  MoveL 2939 to (264.24, 330.75, -7.5) mm, rotated rx 180 ry 0 rz -180 deg; joints [-12.648, -42.636, 107.245, 166.05, 65.267, -174.067]
  MoveL 2940 to (259.09, 331.49, -7.5) mm, rotated rx 180 ry 0 rz 180 deg; joints [-12.718, -42.745, 107.572, 165.997, 65.486, -174.093]
  MoveL 2941 to (253.9, 331.91, -7.5) mm, rotated rx -180 ry 0 rz 180 deg; joints [-12.777, -42.855, 107.905, 165.957, 65.708, -174.125]
  MoveL 2942 to (248.7, 331.99, -7.5) mm, rotated rx -180 ry 0 rz -180 deg; joints [-12.824, -42.967, 108.243, 165.931, 65.932, -174.164]
  MoveL 2943 to (243.5, 331.74, -7.5) mm, rotated rx -180 ry 0 rz 180 deg; joints [-12.859, -43.079, 108.585, 165.917, 66.159, -174.21]
  MoveL 2944 to (238.33, 331.17, -7.5) mm, rotated rx -180 ry 0 rz -180 deg; joints [-12.882, -43.192, 108.929, 165.917, 66.386, -174.262]
  MoveL 2945 to (233.21, 330.26, -7.5) mm, rotated rx 180 ry 0 rz 180 deg; joints [-12.892, -43.304, 109.274, 165.931, 66.613, -174.319]
  MoveL 2946 to (228.15, 329.04, -7.5) mm, rotated rx -180 ry 0 rz 180 deg; joints [-12.89, -43.415, 109.619, 165.958, 66.839, -174.382]
  MoveL 2947 to (223.18, 327.49, -7.5) mm, rotated rx -180 ry 0 rz -180 deg; joints [-12.874, -43.525, 109.963, 165.999, 67.064, -174.45]
  MoveL 2948 to (218.32, 325.63, -7.5) mm, rotated rx 180 ry 0 rz -180 deg; joints [-12.846, -43.634, 110.303, 166.053, 67.286, -174.523]
  MoveL 2949 to (213.59, 323.47, -7.5) mm, rotated rx 180 ry 0 rz -180 deg; joints [-12.804, -43.741, 110.638, 166.121, 67.504, -174.599]
  MoveL 2950 to (209, 321.01, -7.5) mm, rotated rx 180 ry 0 rz 180 deg; joints [-12.75, -43.845, 110.968, 166.202, 67.718, -174.68]
  MoveL 2951 to (204.58, 318.27, -7.5) mm, rotated rx -180 ry 0 rz 180 deg; joints [-12.683, -43.946, 111.291, 166.296, 67.927, -174.764]
  MoveL 2952 to (200.34, 315.25, -7.5) mm, rotated rx -180 ry 0 rz -180 deg; joints [-12.603, -44.044, 111.605, 166.402, 68.13, -174.851]
  MoveL 2953 to (196.3, 311.97, -7.5) mm, rotated rx 180 ry 0 rz 180 deg; joints [-12.51, -44.138, 111.909, 166.521, 68.326, -174.941]
  MoveL 2954 to (192.48, 308.44, -7.5) mm, rotated rx -180 ry 0 rz 180 deg; joints [-12.406, -44.228, 112.202, 166.651, 68.515, -175.033]
  MoveL 2955 to (188.89, 304.68, -7.5) mm, rotated rx -180 ry 0 rz 180 deg; joints [-12.29, -44.314, 112.483, 166.793, 68.694, -175.126]
  MoveL 2956 to (185.54, 300.69, -7.5) mm, rotated rx -180 ry 0 rz -180 deg; joints [-12.162, -44.395, 112.751, 166.946, 68.865, -175.221]
  MoveL 2957 to (182.46, 296.5, -7.5) mm, rotated rx -180 ry 0 rz 180 deg; joints [-12.023, -44.472, 113.004, 167.11, 69.025, -175.317]
  MoveL 2958 to (179.65, 292.12, -7.5) mm, rotated rx 180 ry 0 rz -180 deg; joints [-11.874, -44.543, 113.241, 167.283, 69.175, -175.413]
  MoveL 2959 to (177.12, 287.57, -7.5) mm, rotated rx 180 ry 0 rz -180 deg; joints [-11.715, -44.61, 113.461, 167.465, 69.313, -175.509]
  MoveL 2960 to (174.88, 282.88, -7.5) mm, rotated rx -180 ry 0 rz 180 deg; joints [-11.547, -44.67, 113.664, 167.656, 69.439, -175.605]
  MoveL 2961 to (172.95, 278.05, -7.5) mm, rotated rx -180 ry 0 rz 180 deg; joints [-11.37, -44.725, 113.849, 167.854, 69.552, -175.7]
  MoveL 2962 to (171.32, 273.1, -7.5) mm, rotated rx -180 ry 0 rz -180 deg; joints [-11.186, -44.774, 114.014, 168.059, 69.652, -175.794]
  MoveL 2963 to (170.01, 268.07, -7.5) mm, rotated rx -180 ry 0 rz 180 deg; joints [-10.995, -44.816, 114.159, 168.27, 69.738, -175.887]
  MoveL 2964 to (169.03, 262.96, -7.5) mm, rotated rx 180 ry 0 rz 180 deg; joints [-10.798, -44.853, 114.283, 168.486, 69.81, -175.978]
  MoveL 2965 to (168.37, 257.79, -7.5) mm, rotated rx 180 ry 0 rz -180 deg; joints [-10.596, -44.883, 114.387, 168.706, 69.868, -176.068]
  MoveL 2966 to (168.04, 252.6, -7.5) mm, rotated rx 180 ry 0 rz -180 deg; joints [-10.389, -44.907, 114.468, 168.929, 69.911, -176.155]
  MoveL 2967 to (168.04, 247.4, -7.5) mm, rotated rx 180 ry 0 rz 180 deg; joints [-10.18, -44.925, 114.528, 169.155, 69.938, -176.24]
  MoveL 2968 to (168.37, 242.21, -7.5) mm, rotated rx -180 ry 0 rz -180 deg; joints [-9.968, -44.936, 114.565, 169.381, 69.951, -176.322]
  MoveL 2969 to (169.03, 237.04, -7.5) mm, rotated rx 180 ry 0 rz 180 deg; joints [-9.755, -44.94, 114.581, 169.608, 69.948, -176.402]
  MoveL 2970 to (170.01, 231.93, -7.5) mm, rotated rx 180 ry 0 rz -180 deg; joints [-9.542, -44.938, 114.573, 169.834, 69.929, -176.479]
  MoveL 2971 to (171.32, 226.9, -7.5) mm, rotated rx -180 ry 0 rz 180 deg; joints [-9.33, -44.929, 114.543, 170.058, 69.896, -176.552]
  MoveL 2972 to (172.95, 221.95, -7.5) mm, rotated rx -180 ry 0 rz 180 deg; joints [-9.12, -44.914, 114.491, 170.28, 69.847, -176.623]
  MoveL 2973 to (174.88, 217.12, -7.5) mm, rotated rx 180 ry 0 rz -180 deg; joints [-8.912, -44.892, 114.417, 170.497, 69.783, -176.689]
  MoveL 2974 to (177.12, 212.43, -7.5) mm, rotated rx -180 ry 0 rz 180 deg; joints [-8.709, -44.864, 114.321, 170.71, 69.704, -176.753]
  MoveL 2975 to (179.65, 207.88, -7.5) mm, rotated rx -180 ry 0 rz -180 deg; joints [-8.51, -44.83, 114.204, 170.917, 69.611, -176.812]
  MoveL 2976 to (182.46, 203.5, -7.5) mm, rotated rx -180 ry 0 rz -180 deg; joints [-8.316, -44.789, 114.066, 171.117, 69.505, -176.868]
  MoveL 2977 to (185.54, 199.31, -7.5) mm, rotated rx -180 ry 0 rz 180 deg; joints [-8.13, -44.742, 113.908, 171.31, 69.384, -176.92]
  MoveL 2978 to (188.89, 195.32, -7.5) mm, rotated rx -180 ry 0 rz -180 deg; joints [-7.95, -44.69, 113.73, 171.494, 69.251, -176.967]
  MoveL 2979 to (192.48, 191.56, -7.5) mm, rotated rx -180 ry 0 rz -180 deg; joints [-7.779, -44.631, 113.533, 171.669, 69.106, -177.01]
  MoveL 2980 to (196.3, 188.03, -7.5) mm, rotated rx -180 ry 0 rz -180 deg; joints [-7.617, -44.567, 113.319, 171.835, 68.948, -177.049]
  MoveL 2981 to (200.34, 184.75, -7.5) mm, rotated rx -180 ry 0 rz -180 deg; joints [-7.465, -44.497, 113.087, 171.989, 68.78, -177.084]
  MoveL 2982 to (204.58, 181.73, -7.5) mm, rotated rx -180 ry 0 rz 180 deg; joints [-7.322, -44.422, 112.84, 172.132, 68.602, -177.114]
  MoveL 2983 to (209, 178.99, -7.5) mm, rotated rx -180 ry 0 rz 180 deg; joints [-7.191, -44.343, 112.577, 172.264, 68.414, -177.139]
  MoveL 2984 to (213.59, 176.53, -7.5) mm, rotated rx -180 ry 0 rz -180 deg; joints [-7.07, -44.258, 112.301, 172.383, 68.218, -177.159]
  MoveL 2985 to (218.32, 174.37, -7.5) mm, rotated rx -180 ry 0 rz -180 deg; joints [-6.962, -44.169, 112.012, 172.489, 68.014, -177.174]
  MoveL 2986 to (223.18, 172.51, -7.5) mm, rotated rx 180 ry 0 rz -180 deg; joints [-6.865, -44.077, 111.711, 172.583, 67.804, -177.184]
  MoveL 2987 to (228.15, 170.96, -7.5) mm, rotated rx -180 ry 0 rz -180 deg; joints [-6.781, -43.98, 111.4, 172.662, 67.587, -177.189]
  MoveL 2988 to (233.21, 169.74, -7.5) mm, rotated rx -180 ry 0 rz 180 deg; joints [-6.709, -43.88, 111.081, 172.728, 67.366, -177.188]
  MoveL 2989 to (238.33, 168.83, -7.5) mm, rotated rx 180 ry 0 rz -180 deg; joints [-6.65, -43.777, 110.753, 172.78, 67.14, -177.182]
  MoveL 2990 to (243.5, 168.26, -7.5) mm, rotated rx 180 ry 0 rz -180 deg; joints [-6.605, -43.671, 110.419, 172.817, 66.911, -177.171]
  MoveL 2991 to (248.7, 168.01, -7.5) mm, rotated rx -180 ry 0 rz -180 deg; joints [-6.572, -43.563, 110.08, 172.841, 66.681, -177.154]
  MoveL 2992 to (253.9, 168.09, -7.5) mm, rotated rx 180 ry 0 rz -180 deg; joints [-6.552, -43.453, 109.738, 172.85, 66.449, -177.131]
  MoveL 2993 to (259.09, 168.51, -7.5) mm, rotated rx -180 ry 0 rz 180 deg; joints [-6.545, -43.342, 109.394, 172.845, 66.217, -177.102]
  MoveL 2994 to (264.24, 169.25, -7.5) mm, rotated rx 180 ry 0 rz 180 deg; joints [-6.55, -43.23, 109.048, 172.826, 65.986, -177.068]
  MoveL 2995 to (269.33, 170.31, -7.5) mm, rotated rx -180 ry 0 rz -180 deg; joints [-6.569, -43.118, 108.703, 172.793, 65.756, -177.027]
  MoveL 2996 to (274.35, 171.7, -7.5) mm, rotated rx 180 ry 0 rz -180 deg; joints [-6.6, -43.006, 108.36, 172.746, 65.529, -176.982]
  MoveL 2997 to (279.26, 173.4, -7.5) mm, rotated rx 180 ry 0 rz 180 deg; joints [-6.643, -42.894, 108.021, 172.685, 65.305, -176.93]
  MoveL 2998 to (284.06, 175.41, -7.5) mm, rotated rx -180 ry 0 rz -180 deg; joints [-6.697, -42.783, 107.686, 172.612, 65.086, -176.873]
  MoveL 2999 to (288.73, 177.72, -7.5) mm, rotated rx 180 ry 0 rz 180 deg; joints [-6.764, -42.673, 107.357, 172.525, 64.872, -176.811]
  MoveL 3000 to (293.23, 180.32, -7.5) mm, rotated rx -180 ry 0 rz -180 deg; joints [-6.842, -42.565, 107.035, 172.426, 64.665, -176.744]
  MoveL 3001 to (297.56, 183.2, -7.5) mm, rotated rx 180 ry 0 rz -180 deg; joints [-6.93, -42.46, 106.722, 172.315, 64.464, -176.671]
  MoveL 3002 to (301.71, 186.36, -7.5) mm, rotated rx 180 ry 0 rz 180 deg; joints [-7.029, -42.358, 106.418, 172.193, 64.27, -176.594]
  MoveL 3003 to (305.64, 189.76, -7.5) mm, rotated rx -180 ry 0 rz -180 deg; joints [-7.138, -42.258, 106.126, 172.059, 64.085, -176.512]
  MoveL 3004 to (309.35, 193.41, -7.5) mm, rotated rx 180 ry 0 rz -180 deg; joints [-7.256, -42.163, 105.845, 171.915, 63.909, -176.425]
  MoveL 3005 to (312.82, 197.29, -7.5) mm, rotated rx 180 ry 0 rz 180 deg; joints [-7.383, -42.071, 105.578, 171.762, 63.743, -176.335]
  MoveL 3006 to (316.03, 201.38, -7.5) mm, rotated rx 180 ry 0 rz 180 deg; joints [-7.519, -41.985, 105.325, 171.599, 63.587, -176.241]
  MoveL 3007 to (318.98, 205.67, -7.5) mm, rotated rx -180 ry 0 rz -180 deg; joints [-7.663, -41.903, 105.087, 171.427, 63.443, -176.144]
  MoveL 3008 to (321.66, 210.13, -7.5) mm, rotated rx -180 ry 0 rz -180 deg; joints [-7.813, -41.826, 104.865, 171.248, 63.309, -176.044]
  MoveL 3009 to (324.04, 214.76, -7.5) mm, rotated rx 180 ry 0 rz -180 deg; joints [-7.971, -41.755, 104.66, 171.062, 63.188, -175.942]
  MoveL 3010 to (326.13, 219.52, -7.5) mm, rotated rx -180 ry 0 rz -180 deg; joints [-8.134, -41.69, 104.473, 170.869, 63.079, -175.838]
  MoveL 3011 to (327.91, 224.41, -7.5) mm, rotated rx 180 ry 0 rz 180 deg; joints [-8.304, -41.632, 104.304, 170.671, 62.983, -175.732]
  MoveL 3012 to (329.37, 229.41, -7.5) mm, rotated rx 180 ry 0 rz 180 deg; joints [-8.478, -41.58, 104.155, 170.467, 62.9, -175.625]
  MoveL 3013 to (330.52, 234.48, -7.5) mm, rotated rx 180 ry 0 rz -180 deg; joints [-8.656, -41.534, 104.025, 170.26, 62.83, -175.518]
  MoveL 3014 to (331.34, 239.62, -7.5) mm, rotated rx 180 ry 0 rz -180 deg; joints [-8.838, -41.496, 103.916, 170.05, 62.774, -175.411]
  MoveL 3015 to (331.83, 244.8, -7.5) mm, rotated rx 180 ry 0 rz 180 deg; joints [-9.023, -41.465, 103.827, 169.837, 62.732, -175.305]
  MoveL 3016 to (332, 250, -7.5) mm, rotated rx -180 ry 0 rz 180 deg; joints [-9.211, -41.441, 103.759, 169.623, 62.705, -175.2]
  MoveL 3017 to (320, 250, -7.5) mm, rotated rx -180 ry 0 rz 180 deg; joints [-9.282, -41.725, 104.572, 169.592, 63.231, -175.271]
  MoveL 3018 to (319.86, 254.44, -7.5) mm, rotated rx -180 ry 0 rz -180 deg; joints [-9.445, -41.711, 104.532, 169.408, 63.219, -175.184]
  MoveL 3019 to (319.44, 258.86, -7.5) mm, rotated rx 180 ry 0 rz -180 deg; joints [-9.608, -41.703, 104.51, 169.224, 63.219, -175.099]
  MoveL 3020 to (318.73, 263.25, -7.5) mm, rotated rx 180 ry 0 rz 180 deg; joints [-9.772, -41.702, 104.507, 169.041, 63.231, -175.016]
  MoveL 3021 to (317.76, 267.58, -7.5) mm, rotated rx 180 ry 0 rz 180 deg; joints [-9.936, -41.707, 104.522, 168.859, 63.255, -174.935]
  MoveL 3022 to (316.51, 271.84, -7.5) mm, rotated rx -180 ry 0 rz -180 deg; joints [-10.099, -41.719, 104.556, 168.679, 63.291, -174.858]
  MoveL 3023 to (314.99, 276.02, -7.5) mm, rotated rx -180 ry 0 rz 180 deg; joints [-10.261, -41.737, 104.608, 168.502, 63.339, -174.785]
  MoveL 3024 to (313.2, 280.09, -7.5) mm, rotated rx 180 ry 0 rz 180 deg; joints [-10.421, -41.761, 104.678, 168.329, 63.399, -174.715]
  MoveL 3025 to (311.17, 284.03, -7.5) mm, rotated rx 180 ry 0 rz -180 deg; joints [-10.579, -41.792, 104.765, 168.159, 63.469, -174.65]
  MoveL 3026 to (308.89, 287.84, -7.5) mm, rotated rx -180 ry 0 rz 180 deg; joints [-10.733, -41.828, 104.87, 167.995, 63.551, -174.589]
  MoveL 3027 to (306.37, 291.5, -7.5) mm, rotated rx 180 ry 0 rz 180 deg; joints [-10.884, -41.87, 104.993, 167.835, 63.644, -174.533]
  MoveL 3028 to (303.62, 295, -7.5) mm, rotated rx -180 ry 0 rz 180 deg; joints [-11.03, -41.918, 105.131, 167.682, 63.746, -174.483]
  MoveL 3029 to (300.66, 298.31, -7.5) mm, rotated rx 180 ry 0 rz 180 deg; joints [-11.172, -41.971, 105.286, 167.535, 63.859, -174.437]
  MoveL 3030 to (297.5, 301.42, -7.5) mm, rotated rx 180 ry 0 rz -180 deg; joints [-11.309, -42.03, 105.456, 167.395, 63.981, -174.398]
  MoveL 3031 to (294.14, 304.33, -7.5) mm, rotated rx 180 ry 0 rz -180 deg; joints [-11.44, -42.093, 105.641, 167.263, 64.113, -174.364]
  MoveL 3032 to (290.6, 307.02, -7.5) mm, rotated rx 180 ry 0 rz -180 deg; joints [-11.565, -42.161, 105.84, 167.139, 64.253, -174.336]
  MoveL 3033 to (286.91, 309.48, -7.5) mm, rotated rx 180 ry 0 rz -180 deg; joints [-11.683, -42.233, 106.052, 167.024, 64.401, -174.314]
  MoveL 3034 to (283.06, 311.7, -7.5) mm, rotated rx 180 ry 0 rz -180 deg; joints [-11.794, -42.309, 106.276, 166.917, 64.556, -174.299]
  MoveL 3035 to (279.08, 313.67, -7.5) mm, rotated rx 180 ry 0 rz -180 deg; joints [-11.898, -42.389, 106.512, 166.82, 64.719, -174.289]
  MoveL 3036 to (274.98, 315.39, -7.5) mm, rotated rx 180 ry 0 rz 180 deg; joints [-11.993, -42.472, 106.759, 166.733, 64.887, -174.286]
  MoveL 3037 to (270.78, 316.84, -7.5) mm, rotated rx 180 ry 0 rz -180 deg; joints [-12.08, -42.559, 107.015, 166.656, 65.061, -174.289]
  MoveL 3038 to (266.5, 318.03, -7.5) mm, rotated rx 180 ry 0 rz -180 deg; joints [-12.158, -42.647, 107.28, 166.59, 65.24, -174.298]
  MoveL 3039 to (262.16, 318.94, -7.5) mm, rotated rx -180 ry 0 rz -180 deg; joints [-12.226, -42.738, 107.553, 166.534, 65.424, -174.313]
  MoveL 3040 to (257.76, 319.57, -7.5) mm, rotated rx 180 ry 0 rz 180 deg; joints [-12.285, -42.831, 107.832, 166.489, 65.611, -174.334]
  MoveL 3041 to (253.33, 319.92, -7.5) mm, rotated rx -180 ry 0 rz -180 deg; joints [-12.335, -42.925, 108.116, 166.455, 65.801, -174.36]
  MoveL 3042 to (248.89, 319.99, -7.5) mm, rotated rx 180 ry 0 rz 180 deg; joints [-12.374, -43.02, 108.405, 166.433, 65.993, -174.393]
  MoveL 3043 to (244.45, 319.78, -7.5) mm, rotated rx 180 ry 0 rz -180 deg; joints [-12.402, -43.116, 108.697, 166.422, 66.187, -174.431]
  MoveL 3044 to (240.04, 319.29, -7.5) mm, rotated rx 180 ry 0 rz 180 deg; joints [-12.42, -43.212, 108.991, 166.423, 66.381, -174.474]
  MoveL 3045 to (235.66, 318.52, -7.5) mm, rotated rx -180 ry 0 rz 180 deg; joints [-12.428, -43.308, 109.286, 166.436, 66.575, -174.521]
  MoveL 3046 to (231.35, 317.47, -7.5) mm, rotated rx 180 ry 0 rz -180 deg; joints [-12.424, -43.403, 109.581, 166.46, 66.769, -174.574]
  MoveL 3047 to (227.11, 316.15, -7.5) mm, rotated rx 180 ry 0 rz -180 deg; joints [-12.409, -43.497, 109.874, 166.495, 66.961, -174.631]
  MoveL 3048 to (222.96, 314.56, -7.5) mm, rotated rx 180 ry 0 rz -180 deg; joints [-12.384, -43.59, 110.164, 166.543, 67.15, -174.691]
  MoveL 3049 to (218.92, 312.72, -7.5) mm, rotated rx -180 ry 0 rz 180 deg; joints [-12.347, -43.681, 110.45, 166.601, 67.337, -174.756]
  MoveL 3050 to (215, 310.62, -7.5) mm, rotated rx 180 ry 0 rz 180 deg; joints [-12.299, -43.77, 110.731, 166.671, 67.52, -174.824]
  MoveL 3051 to (211.23, 308.28, -7.5) mm, rotated rx -180 ry 0 rz 180 deg; joints [-12.241, -43.857, 111.007, 166.752, 67.698, -174.894]
  MoveL 3052 to (207.61, 305.7, -7.5) mm, rotated rx 180 ry 0 rz 180 deg; joints [-12.172, -43.941, 111.274, 166.844, 67.871, -174.968]
  MoveL 3053 to (204.16, 302.9, -7.5) mm, rotated rx 180 ry 0 rz -180 deg; joints [-12.092, -44.021, 111.534, 166.946, 68.038, -175.044]
  MoveL 3054 to (200.9, 299.89, -7.5) mm, rotated rx -180 ry 0 rz 180 deg; joints [-12.002, -44.099, 111.783, 167.058, 68.198, -175.122]
  MoveL 3055 to (197.83, 296.67, -7.5) mm, rotated rx -180 ry 0 rz 180 deg; joints [-11.902, -44.173, 112.023, 167.179, 68.351, -175.201]
  MoveL 3056 to (194.98, 293.27, -7.5) mm, rotated rx 180 ry 0 rz -180 deg; joints [-11.793, -44.243, 112.251, 167.311, 68.495, -175.281]
  MoveL 3057 to (192.34, 289.69, -7.5) mm, rotated rx 180 ry 0 rz 180 deg; joints [-11.674, -44.309, 112.466, 167.45, 68.631, -175.363]
  MoveL 3058 to (189.94, 285.96, -7.5) mm, rotated rx 180 ry 0 rz -180 deg; joints [-11.547, -44.37, 112.668, 167.598, 68.758, -175.445]
  MoveL 3059 to (187.78, 282.08, -7.5) mm, rotated rx -180 ry 0 rz -180 deg; joints [-11.412, -44.427, 112.855, 167.754, 68.875, -175.527]
  MoveL 3060 to (185.87, 278.07, -7.5) mm, rotated rx -180 ry 0 rz -180 deg; joints [-11.269, -44.479, 113.028, 167.917, 68.982, -175.609]
  MoveL 3061 to (184.22, 273.94, -7.5) mm, rotated rx -180 ry 0 rz 180 deg; joints [-11.118, -44.527, 113.185, 168.086, 69.078, -175.691]
  MoveL 3062 to (182.84, 269.72, -7.5) mm, rotated rx 180 ry 0 rz 180 deg; joints [-10.962, -44.569, 113.325, 168.26, 69.162, -175.772]
  MoveL 3063 to (181.72, 265.42, -7.5) mm, rotated rx 180 ry 0 rz 180 deg; joints [-10.8, -44.606, 113.449, 168.44, 69.235, -175.852]
  MoveL 3064 to (180.88, 261.06, -7.5) mm, rotated rx 180 ry 0 rz 180 deg; joints [-10.633, -44.637, 113.555, 168.624, 69.296, -175.931]
  MoveL 3065 to (180.32, 256.65, -7.5) mm, rotated rx -180 ry 0 rz -180 deg; joints [-10.461, -44.664, 113.643, 168.811, 69.345, -176.009]
  MoveL 3066 to (180.04, 252.22, -7.5) mm, rotated rx 180 ry 0 rz 180 deg; joints [-10.287, -44.684, 113.712, 169.001, 69.38, -176.084]
  MoveL 3067 to (180.04, 247.78, -7.5) mm, rotated rx 180 ry 0 rz -180 deg; joints [-10.109, -44.699, 113.763, 169.193, 69.403, -176.158]
  MoveL 3068 to (180.32, 243.35, -7.5) mm, rotated rx -180 ry 0 rz -180 deg; joints [-9.93, -44.709, 113.795, 169.385, 69.414, -176.23]
  MoveL 3069 to (180.88, 238.94, -7.5) mm, rotated rx 180 ry 0 rz 180 deg; joints [-9.75, -44.713, 113.808, 169.578, 69.411, -176.299]
  MoveL 3070 to (181.72, 234.58, -7.5) mm, rotated rx -180 ry 0 rz 180 deg; joints [-9.569, -44.711, 113.801, 169.77, 69.395, -176.366]
  MoveL 3071 to (182.84, 230.28, -7.5) mm, rotated rx -180 ry 0 rz 180 deg; joints [-9.39, -44.703, 113.776, 169.96, 69.366, -176.43]
  MoveL 3072 to (184.22, 226.06, -7.5) mm, rotated rx 180 ry 0 rz 180 deg; joints [-9.212, -44.69, 113.732, 170.148, 69.324, -176.491]
  MoveL 3073 to (185.87, 221.93, -7.5) mm, rotated rx -180 ry 0 rz 180 deg; joints [-9.036, -44.671, 113.669, 170.333, 69.27, -176.549]
  MoveL 3074 to (187.78, 217.92, -7.5) mm, rotated rx 180 ry 0 rz 180 deg; joints [-8.863, -44.647, 113.587, 170.513, 69.203, -176.605]
  MoveL 3075 to (189.94, 214.04, -7.5) mm, rotated rx -180 ry 0 rz 180 deg; joints [-8.695, -44.617, 113.487, 170.689, 69.124, -176.656]
  MoveL 3076 to (192.34, 210.31, -7.5) mm, rotated rx -180 ry 0 rz 180 deg; joints [-8.531, -44.582, 113.37, 170.859, 69.034, -176.705]
  MoveL 3077 to (194.98, 206.73, -7.5) mm, rotated rx 180 ry 0 rz -180 deg; joints [-8.372, -44.542, 113.235, 171.023, 68.932, -176.75]
  MoveL 3078 to (197.83, 203.33, -7.5) mm, rotated rx 180 ry 0 rz -180 deg; joints [-8.22, -44.496, 113.084, 171.18, 68.818, -176.791]
  MoveL 3079 to (200.9, 200.11, -7.5) mm, rotated rx 180 ry 0 rz 180 deg; joints [-8.074, -44.446, 112.917, 171.329, 68.695, -176.829]
  MoveL 3080 to (204.16, 197.1, -7.5) mm, rotated rx -180 ry 0 rz -180 deg; joints [-7.936, -44.39, 112.734, 171.47, 68.562, -176.862]
  MoveL 3081 to (207.61, 194.3, -7.5) mm, rotated rx 180 ry 0 rz -180 deg; joints [-7.806, -44.33, 112.537, 171.601, 68.419, -176.892]
  MoveL 3082 to (211.23, 191.72, -7.5) mm, rotated rx 180 ry 0 rz 180 deg; joints [-7.684, -44.266, 112.326, 171.724, 68.267, -176.917]
  MoveL 3083 to (215, 189.38, -7.5) mm, rotated rx -180 ry 0 rz 180 deg; joints [-7.572, -44.197, 112.103, 171.836, 68.108, -176.938]
  MoveL 3084 to (218.92, 187.28, -7.5) mm, rotated rx -180 ry 0 rz -180 deg; joints [-7.468, -44.125, 111.867, 171.938, 67.941, -176.955]
  MoveL 3085 to (222.96, 185.44, -7.5) mm, rotated rx -180 ry 0 rz -180 deg; joints [-7.375, -44.049, 111.621, 172.029, 67.768, -176.967]
  MoveL 3086 to (227.11, 183.85, -7.5) mm, rotated rx -180 ry 0 rz 180 deg; joints [-7.292, -43.969, 111.365, 172.109, 67.589, -176.975]
  MoveL 3087 to (231.35, 182.53, -7.5) mm, rotated rx -180 ry 0 rz -180 deg; joints [-7.219, -43.886, 111.1, 172.177, 67.405, -176.978]
  MoveL 3088 to (235.66, 181.48, -7.5) mm, rotated rx -180 ry 0 rz 180 deg; joints [-7.157, -43.8, 110.827, 172.234, 67.216, -176.977]
  MoveL 3089 to (240.04, 180.71, -7.5) mm, rotated rx -180 ry 0 rz -180 deg; joints [-7.105, -43.712, 110.548, 172.279, 67.024, -176.971]
  MoveL 3090 to (244.45, 180.22, -7.5) mm, rotated rx -180 ry 0 rz -180 deg; joints [-7.065, -43.621, 110.263, 172.312, 66.829, -176.959]
  MoveL 3091 to (248.89, 180.01, -7.5) mm, rotated rx -180 ry 0 rz 180 deg; joints [-7.035, -43.529, 109.974, 172.332, 66.633, -176.943]
  MoveL 3092 to (253.33, 180.08, -7.5) mm, rotated rx -180 ry 0 rz -180 deg; joints [-7.017, -43.435, 109.682, 172.341, 66.435, -176.923]
  MoveL 3093 to (257.76, 180.43, -7.5) mm, rotated rx 180 ry 0 rz 180 deg; joints [-7.01, -43.341, 109.388, 172.337, 66.237, -176.897]
  MoveL 3094 to (262.16, 181.06, -7.5) mm, rotated rx 180 ry 0 rz 180 deg; joints [-7.013, -43.245, 109.093, 172.322, 66.04, -176.866]
  MoveL 3095 to (266.5, 181.97, -7.5) mm, rotated rx -180 ry 0 rz -180 deg; joints [-7.027, -43.149, 108.799, 172.294, 65.844, -176.831]
  MoveL 3096 to (270.78, 183.16, -7.5) mm, rotated rx -180 ry 0 rz -180 deg; joints [-7.052, -43.053, 108.506, 172.255, 65.65, -176.79]
  MoveL 3097 to (274.98, 184.61, -7.5) mm, rotated rx 180 ry 0 rz -180 deg; joints [-7.088, -42.958, 108.216, 172.204, 65.459, -176.745]
  MoveL 3098 to (279.08, 186.33, -7.5) mm, rotated rx -180 ry 0 rz -180 deg; joints [-7.134, -42.863, 107.929, 172.142, 65.272, -176.696]
  MoveL 3099 to (283.06, 188.3, -7.5) mm, rotated rx 180 ry 0 rz -180 deg; joints [-7.189, -42.77, 107.648, 172.069, 65.089, -176.642]
  MoveL 3100 to (286.91, 190.52, -7.5) mm, rotated rx 180 ry 0 rz 180 deg; joints [-7.255, -42.679, 107.373, 171.985, 64.912, -176.583]
  MoveL 3101 to (290.6, 192.98, -7.5) mm, rotated rx -180 ry 0 rz 180 deg; joints [-7.33, -42.589, 107.106, 171.891, 64.74, -176.52]
  MoveL 3102 to (294.14, 195.67, -7.5) mm, rotated rx 180 ry 0 rz 180 deg; joints [-7.413, -42.502, 106.846, 171.786, 64.574, -176.454]
  MoveL 3103 to (297.5, 198.58, -7.5) mm, rotated rx 180 ry 0 rz -180 deg; joints [-7.506, -42.418, 106.596, 171.673, 64.416, -176.383]
  MoveL 3104 to (300.66, 201.69, -7.5) mm, rotated rx -180 ry 0 rz -180 deg; joints [-7.606, -42.337, 106.356, 171.55, 64.265, -176.309]
  MoveL 3105 to (303.62, 205, -7.5) mm, rotated rx -180 ry 0 rz 180 deg; joints [-7.715, -42.259, 106.128, 171.419, 64.123, -176.232]
  MoveL 3106 to (306.37, 208.5, -7.5) mm, rotated rx -180 ry 0 rz -180 deg; joints [-7.83, -42.185, 105.911, 171.281, 63.989, -176.152]
  MoveL 3107 to (308.89, 212.16, -7.5) mm, rotated rx -180 ry 0 rz -180 deg; joints [-7.953, -42.116, 105.708, 171.134, 63.865, -176.07]
  MoveL 3108 to (311.17, 215.97, -7.5) mm, rotated rx 180 ry 0 rz -180 deg; joints [-8.082, -42.051, 105.518, 170.981, 63.751, -175.985]
  MoveL 3109 to (313.2, 219.91, -7.5) mm, rotated rx -180 ry 0 rz 180 deg; joints [-8.217, -41.991, 105.343, 170.822, 63.647, -175.898]
  MoveL 3110 to (314.99, 223.98, -7.5) mm, rotated rx -180 ry 0 rz 180 deg; joints [-8.357, -41.936, 105.183, 170.658, 63.553, -175.809]
  MoveL 3111 to (316.51, 228.16, -7.5) mm, rotated rx 180 ry 0 rz -180 deg; joints [-8.502, -41.886, 105.039, 170.488, 63.471, -175.72]
  MoveL 3112 to (317.76, 232.42, -7.5) mm, rotated rx 180 ry 0 rz -180 deg; joints [-8.652, -41.842, 104.911, 170.315, 63.4, -175.63]
  MoveL 3113 to (318.73, 236.75, -7.5) mm, rotated rx 180 ry 0 rz 180 deg; joints [-8.805, -41.804, 104.8, 170.138, 63.34, -175.54]
  MoveL 3114 to (319.44, 241.14, -7.5) mm, rotated rx 180 ry 0 rz -180 deg; joints [-8.962, -41.771, 104.706, 169.958, 63.292, -175.449]
  MoveL 3115 to (319.86, 245.56, -7.5) mm, rotated rx 180 ry 0 rz 180 deg; joints [-9.121, -41.745, 104.63, 169.776, 63.255, -175.36]
  MoveL 3116 to (320, 250, -7.5) mm, rotated rx -180 ry 0 rz 180 deg; joints [-9.282, -41.725, 104.572, 169.592, 63.231, -175.271]
  MoveL 3117 to (308, 250, -7.5) mm, rotated rx -180 ry 0 rz -180 deg; joints [-9.354, -42.004, 105.38, 169.56, 63.758, -175.342]
  MoveL 3118 to (307.88, 253.68, -7.5) mm, rotated rx -180 ry 0 rz -180 deg; joints [-9.49, -41.992, 105.347, 169.407, 63.748, -175.271]
  MoveL 3119 to (307.53, 257.34, -7.5) mm, rotated rx 180 ry 0 rz 180 deg; joints [-9.626, -41.986, 105.329, 169.254, 63.747, -175.201]
  MoveL 3120 to (306.95, 260.98, -7.5) mm, rotated rx -180 ry 0 rz -180 deg; joints [-9.764, -41.985, 105.327, 169.102, 63.757, -175.134]
  MoveL 3121 to (306.14, 264.57, -7.5) mm, rotated rx 180 ry 0 rz -180 deg; joints [-9.9, -41.99, 105.339, 168.95, 63.777, -175.068]
  MoveL 3122 to (305.1, 268.1, -7.5) mm, rotated rx 180 ry 0 rz -180 deg; joints [-10.037, -41.999, 105.367, 168.801, 63.807, -175.005]
  MoveL 3123 to (303.85, 271.56, -7.5) mm, rotated rx 180 ry 0 rz -180 deg; joints [-10.172, -42.014, 105.41, 168.654, 63.846, -174.945]
  MoveL 3124 to (302.37, 274.93, -7.5) mm, rotated rx -180 ry 0 rz -180 deg; joints [-10.305, -42.034, 105.468, 168.509, 63.896, -174.889]
  MoveL 3125 to (300.68, 278.2, -7.5) mm, rotated rx 180 ry 0 rz 180 deg; joints [-10.436, -42.059, 105.541, 168.368, 63.954, -174.835]
  MoveL 3126 to (298.79, 281.36, -7.5) mm, rotated rx 180 ry 0 rz 180 deg; joints [-10.565, -42.089, 105.628, 168.231, 64.022, -174.786]
  MoveL 3127 to (296.71, 284.39, -7.5) mm, rotated rx 180 ry 0 rz 180 deg; joints [-10.691, -42.123, 105.73, 168.099, 64.099, -174.74]
  MoveL 3128 to (294.43, 287.28, -7.5) mm, rotated rx -180 ry 0 rz -180 deg; joints [-10.813, -42.163, 105.845, 167.971, 64.184, -174.699]
  MoveL 3129 to (291.98, 290.02, -7.5) mm, rotated rx -180 ry 0 rz -180 deg; joints [-10.931, -42.206, 105.973, 167.849, 64.278, -174.661]
  MoveL 3130 to (289.35, 292.61, -7.5) mm, rotated rx 180 ry 0 rz -180 deg; joints [-11.045, -42.254, 106.114, 167.733, 64.38, -174.629]
  MoveL 3131 to (286.57, 295.02, -7.5) mm, rotated rx -180 ry 0 rz -180 deg; joints [-11.154, -42.307, 106.268, 167.623, 64.489, -174.601]
  MoveL 3132 to (283.64, 297.25, -7.5) mm, rotated rx 180 ry 0 rz 180 deg; joints [-11.257, -42.362, 106.433, 167.52, 64.605, -174.578]
  MoveL 3133 to (280.58, 299.28, -7.5) mm, rotated rx 180 ry 0 rz 180 deg; joints [-11.355, -42.422, 106.609, 167.424, 64.728, -174.56]
  MoveL 3134 to (277.39, 301.12, -7.5) mm, rotated rx 180 ry 0 rz -180 deg; joints [-11.447, -42.485, 106.795, 167.336, 64.857, -174.547]
  MoveL 3135 to (274.09, 302.76, -7.5) mm, rotated rx -180 ry 0 rz -180 deg; joints [-11.533, -42.551, 106.991, 167.255, 64.992, -174.538]
  MoveL 3136 to (270.7, 304.18, -7.5) mm, rotated rx -180 ry 0 rz -180 deg; joints [-11.611, -42.619, 107.196, 167.183, 65.133, -174.535]
  MoveL 3137 to (267.22, 305.38, -7.5) mm, rotated rx 180 ry 0 rz 180 deg; joints [-11.682, -42.69, 107.408, 167.119, 65.277, -174.537]
  MoveL 3138 to (263.67, 306.37, -7.5) mm, rotated rx 180 ry 0 rz 180 deg; joints [-11.746, -42.763, 107.628, 167.064, 65.426, -174.544]
  MoveL 3139 to (260.07, 307.12, -7.5) mm, rotated rx -180 ry 0 rz -180 deg; joints [-11.803, -42.838, 107.854, 167.018, 65.579, -174.556]
  MoveL 3140 to (256.43, 307.64, -7.5) mm, rotated rx 180 ry 0 rz -180 deg; joints [-11.851, -42.915, 108.086, 166.982, 65.734, -174.572]
  MoveL 3141 to (252.76, 307.93, -7.5) mm, rotated rx 180 ry 0 rz -180 deg; joints [-11.89, -42.993, 108.322, 166.954, 65.892, -174.593]
  MoveL 3142 to (249.08, 307.99, -7.5) mm, rotated rx 180 ry 0 rz -180 deg; joints [-11.922, -43.071, 108.561, 166.936, 66.052, -174.619]
  MoveL 3143 to (245.4, 307.82, -7.5) mm, rotated rx -180 ry 0 rz 180 deg; joints [-11.944, -43.151, 108.803, 166.928, 66.213, -174.65]
  MoveL 3144 to (241.75, 307.41, -7.5) mm, rotated rx -180 ry 0 rz -180 deg; joints [-11.958, -43.23, 109.047, 166.929, 66.374, -174.684]
  MoveL 3145 to (238.12, 306.77, -7.5) mm, rotated rx 180 ry 0 rz -180 deg; joints [-11.963, -43.309, 109.291, 166.94, 66.535, -174.723]
  MoveL 3146 to (234.54, 305.9, -7.5) mm, rotated rx 180 ry 0 rz -180 deg; joints [-11.959, -43.388, 109.535, 166.961, 66.696, -174.765]
  MoveL 3147 to (231.03, 304.81, -7.5) mm, rotated rx 180 ry 0 rz 180 deg; joints [-11.946, -43.466, 109.778, 166.991, 66.855, -174.811]
  MoveL 3148 to (227.59, 303.5, -7.5) mm, rotated rx 180 ry 0 rz 180 deg; joints [-11.923, -43.543, 110.018, 167.031, 67.012, -174.861]
  MoveL 3149 to (224.24, 301.97, -7.5) mm, rotated rx 180 ry 0 rz 180 deg; joints [-11.892, -43.619, 110.255, 167.08, 67.167, -174.913]
  MoveL 3150 to (221, 300.23, -7.5) mm, rotated rx -180 ry 0 rz -180 deg; joints [-11.851, -43.693, 110.488, 167.139, 67.318, -174.968]
  MoveL 3151 to (217.87, 298.29, -7.5) mm, rotated rx 180 ry 0 rz 180 deg; joints [-11.802, -43.765, 110.716, 167.206, 67.465, -175.026]
  MoveL 3152 to (214.87, 296.15, -7.5) mm, rotated rx -180 ry 0 rz 180 deg; joints [-11.744, -43.835, 110.938, 167.283, 67.608, -175.087]
  MoveL 3153 to (212.02, 293.83, -7.5) mm, rotated rx -180 ry 0 rz 180 deg; joints [-11.677, -43.902, 111.152, 167.368, 67.746, -175.149]
  MoveL 3154 to (209.31, 291.34, -7.5) mm, rotated rx -180 ry 0 rz 180 deg; joints [-11.602, -43.967, 111.359, 167.462, 67.878, -175.213]
  MoveL 3155 to (206.77, 288.67, -7.5) mm, rotated rx 180 ry 0 rz 180 deg; joints [-11.519, -44.029, 111.557, 167.563, 68.005, -175.278]
  MoveL 3156 to (204.41, 285.85, -7.5) mm, rotated rx -180 ry 0 rz -180 deg; joints [-11.428, -44.087, 111.745, 167.672, 68.124, -175.345]
  MoveL 3157 to (202.23, 282.89, -7.5) mm, rotated rx 180 ry 0 rz -180 deg; joints [-11.33, -44.142, 111.923, 167.788, 68.236, -175.412]
  MoveL 3158 to (200.24, 279.79, -7.5) mm, rotated rx 180 ry 0 rz -180 deg; joints [-11.224, -44.193, 112.09, 167.911, 68.341, -175.48]
  MoveL 3159 to (198.45, 276.58, -7.5) mm, rotated rx 180 ry 0 rz 180 deg; joints [-11.112, -44.241, 112.245, 168.04, 68.437, -175.548]
  MoveL 3160 to (196.87, 273.25, -7.5) mm, rotated rx -180 ry 0 rz -180 deg; joints [-10.994, -44.285, 112.388, 168.174, 68.525, -175.617]
  MoveL 3161 to (195.5, 269.84, -7.5) mm, rotated rx -180 ry 0 rz -180 deg; joints [-10.87, -44.324, 112.517, 168.314, 68.603, -175.685]
  MoveL 3162 to (194.35, 266.34, -7.5) mm, rotated rx -180 ry 0 rz -180 deg; joints [-10.741, -44.36, 112.633, 168.459, 68.673, -175.753]
  MoveL 3163 to (193.43, 262.78, -7.5) mm, rotated rx 180 ry 0 rz -180 deg; joints [-10.608, -44.391, 112.735, 168.607, 68.733, -175.82]
  MoveL 3164 to (192.73, 259.16, -7.5) mm, rotated rx 180 ry 0 rz 180 deg; joints [-10.47, -44.417, 112.822, 168.759, 68.782, -175.886]
  MoveL 3165 to (192.26, 255.51, -7.5) mm, rotated rx 180 ry 0 rz 180 deg; joints [-10.329, -44.439, 112.895, 168.914, 68.822, -175.951]
  MoveL 3166 to (192.03, 251.84, -7.5) mm, rotated rx 180 ry 0 rz -180 deg; joints [-10.185, -44.457, 112.952, 169.07, 68.851, -176.015]
  MoveL 3167 to (192.03, 248.16, -7.5) mm, rotated rx 180 ry 0 rz -180 deg; joints [-10.04, -44.469, 112.994, 169.228, 68.87, -176.077]
  MoveL 3168 to (192.26, 244.49, -7.5) mm, rotated rx 180 ry 0 rz 180 deg; joints [-9.892, -44.477, 113.021, 169.387, 68.878, -176.137]
  MoveL 3169 to (192.73, 240.84, -7.5) mm, rotated rx 180 ry 0 rz 180 deg; joints [-9.744, -44.48, 113.031, 169.546, 68.875, -176.196]
  MoveL 3170 to (193.43, 237.22, -7.5) mm, rotated rx -180 ry 0 rz -180 deg; joints [-9.596, -44.479, 113.026, 169.704, 68.862, -176.252]
  MoveL 3171 to (194.35, 233.66, -7.5) mm, rotated rx 180 ry 0 rz 180 deg; joints [-9.448, -44.472, 113.005, 169.861, 68.838, -176.306]
  MoveL 3172 to (195.5, 230.16, -7.5) mm, rotated rx -180 ry 0 rz -180 deg; joints [-9.302, -44.461, 112.969, 170.016, 68.804, -176.358]
  MoveL 3173 to (196.87, 226.75, -7.5) mm, rotated rx -180 ry 0 rz -180 deg; joints [-9.158, -44.446, 112.917, 170.169, 68.759, -176.407]
  MoveL 3174 to (198.45, 223.42, -7.5) mm, rotated rx 180 ry 0 rz 180 deg; joints [-9.016, -44.425, 112.849, 170.317, 68.704, -176.454]
  MoveL 3175 to (200.24, 220.21, -7.5) mm, rotated rx 180 ry 0 rz 180 deg; joints [-8.877, -44.4, 112.767, 170.462, 68.638, -176.498]
  MoveL 3176 to (202.23, 217.11, -7.5) mm, rotated rx 180 ry 0 rz -180 deg; joints [-8.742, -44.371, 112.67, 170.603, 68.564, -176.539]
  MoveL 3177 to (204.41, 214.15, -7.5) mm, rotated rx 180 ry 0 rz -180 deg; joints [-8.611, -44.337, 112.559, 170.738, 68.479, -176.577]
  MoveL 3178 to (206.77, 211.33, -7.5) mm, rotated rx -180 ry 0 rz 180 deg; joints [-8.486, -44.299, 112.434, 170.867, 68.386, -176.611]
  MoveL 3179 to (209.31, 208.66, -7.5) mm, rotated rx -180 ry 0 rz -180 deg; joints [-8.365, -44.257, 112.296, 170.991, 68.285, -176.643]
  MoveL 3180 to (212.02, 206.17, -7.5) mm, rotated rx 180 ry 0 rz 180 deg; joints [-8.251, -44.21, 112.145, 171.107, 68.175, -176.671]
  MoveL 3181 to (214.87, 203.85, -7.5) mm, rotated rx 180 ry 0 rz 180 deg; joints [-8.143, -44.16, 111.982, 171.216, 68.057, -176.695]
  MoveL 3182 to (217.87, 201.71, -7.5) mm, rotated rx 180 ry 0 rz 180 deg; joints [-8.042, -44.106, 111.808, 171.317, 67.932, -176.716]
  MoveL 3183 to (221, 199.77, -7.5) mm, rotated rx 180 ry 0 rz 180 deg; joints [-7.949, -44.049, 111.623, 171.41, 67.801, -176.733]
  MoveL 3184 to (224.24, 198.03, -7.5) mm, rotated rx 180 ry 0 rz -180 deg; joints [-7.863, -43.989, 111.428, 171.495, 67.663, -176.747]
  MoveL 3185 to (227.59, 196.5, -7.5) mm, rotated rx 180 ry 0 rz -180 deg; joints [-7.785, -43.925, 111.224, 171.57, 67.52, -176.757]
  MoveL 3186 to (231.03, 195.19, -7.5) mm, rotated rx -180 ry 0 rz -180 deg; joints [-7.715, -43.858, 111.012, 171.637, 67.372, -176.763]
  MoveL 3187 to (234.54, 194.1, -7.5) mm, rotated rx -180 ry 0 rz -180 deg; joints [-7.654, -43.789, 110.793, 171.694, 67.22, -176.765]
  MoveL 3188 to (238.12, 193.23, -7.5) mm, rotated rx -180 ry 0 rz -180 deg; joints [-7.602, -43.718, 110.568, 171.741, 67.065, -176.763]
  MoveL 3189 to (241.75, 192.59, -7.5) mm, rotated rx 180 ry 0 rz -180 deg; joints [-7.558, -43.645, 110.336, 171.779, 66.906, -176.756]
  MoveL 3190 to (245.4, 192.18, -7.5) mm, rotated rx -180 ry 0 rz -180 deg; joints [-7.524, -43.57, 110.101, 171.807, 66.745, -176.746]
  MoveL 3191 to (249.08, 192.01, -7.5) mm, rotated rx 180 ry 0 rz -180 deg; joints [-7.498, -43.493, 109.861, 171.824, 66.582, -176.732]
  MoveL 3192 to (252.76, 192.07, -7.5) mm, rotated rx 180 ry 0 rz 180 deg; joints [-7.482, -43.415, 109.619, 171.832, 66.419, -176.714]
  MoveL 3193 to (256.43, 192.36, -7.5) mm, rotated rx 180 ry 0 rz 180 deg; joints [-7.475, -43.337, 109.376, 171.83, 66.255, -176.691]
  MoveL 3194 to (260.07, 192.88, -7.5) mm, rotated rx -180 ry 0 rz -180 deg; joints [-7.476, -43.257, 109.131, 171.817, 66.092, -176.665]
  MoveL 3195 to (263.67, 193.63, -7.5) mm, rotated rx 180 ry 0 rz 180 deg; joints [-7.487, -43.178, 108.887, 171.795, 65.93, -176.634]
  MoveL 3196 to (267.22, 194.62, -7.5) mm, rotated rx 180 ry 0 rz -180 deg; joints [-7.507, -43.099, 108.645, 171.763, 65.769, -176.6]
  MoveL 3197 to (270.7, 195.82, -7.5) mm, rotated rx 180 ry 0 rz -180 deg; joints [-7.535, -43.02, 108.404, 171.722, 65.611, -176.562]
  MoveL 3198 to (274.09, 197.24, -7.5) mm, rotated rx -180 ry 0 rz 180 deg; joints [-7.572, -42.942, 108.167, 171.671, 65.455, -176.52]
  MoveL 3199 to (277.39, 198.88, -7.5) mm, rotated rx 180 ry 0 rz 180 deg; joints [-7.617, -42.865, 107.934, 171.611, 65.304, -176.474]
  MoveL 3200 to (280.58, 200.72, -7.5) mm, rotated rx -180 ry 0 rz -180 deg; joints [-7.671, -42.789, 107.706, 171.542, 65.156, -176.425]
  MoveL 3201 to (283.64, 202.75, -7.5) mm, rotated rx 180 ry 0 rz 180 deg; joints [-7.732, -42.715, 107.484, 171.464, 65.013, -176.372]
  MoveL 3202 to (286.57, 204.98, -7.5) mm, rotated rx -180 ry 0 rz -180 deg; joints [-7.801, -42.643, 107.268, 171.378, 64.876, -176.317]
  MoveL 3203 to (289.35, 207.39, -7.5) mm, rotated rx 180 ry 0 rz -180 deg; joints [-7.877, -42.574, 107.061, 171.284, 64.745, -176.258]
  MoveL 3204 to (291.98, 209.98, -7.5) mm, rotated rx 180 ry 0 rz 180 deg; joints [-7.96, -42.507, 106.862, 171.183, 64.619, -176.196]
  MoveL 3205 to (294.43, 212.72, -7.5) mm, rotated rx -180 ry 0 rz 180 deg; joints [-8.05, -42.443, 106.672, 171.075, 64.501, -176.132]
  MoveL 3206 to (296.71, 215.61, -7.5) mm, rotated rx 180 ry 0 rz -180 deg; joints [-8.145, -42.383, 106.492, 170.96, 64.39, -176.066]
  MoveL 3207 to (298.79, 218.64, -7.5) mm, rotated rx -180 ry 0 rz 180 deg; joints [-8.247, -42.325, 106.323, 170.839, 64.287, -175.998]
  MoveL 3208 to (300.68, 221.8, -7.5) mm, rotated rx 180 ry 0 rz -180 deg; joints [-8.354, -42.272, 106.166, 170.712, 64.192, -175.928]
  MoveL 3209 to (302.37, 225.07, -7.5) mm, rotated rx -180 ry 0 rz 180 deg; joints [-8.466, -42.223, 106.021, 170.581, 64.105, -175.856]
  MoveL 3210 to (303.85, 228.44, -7.5) mm, rotated rx 180 ry 0 rz -180 deg; joints [-8.583, -42.177, 105.888, 170.444, 64.027, -175.783]
  MoveL 3211 to (305.1, 231.9, -7.5) mm, rotated rx -180 ry 0 rz -180 deg; joints [-8.704, -42.136, 105.768, 170.304, 63.958, -175.71]
  MoveL 3212 to (306.14, 235.43, -7.5) mm, rotated rx -180 ry 0 rz -180 deg; joints [-8.828, -42.1, 105.662, 170.16, 63.899, -175.636]
  MoveL 3213 to (306.95, 239.02, -7.5) mm, rotated rx -180 ry 0 rz 180 deg; joints [-8.956, -42.069, 105.57, 170.013, 63.849, -175.562]
  MoveL 3214 to (307.53, 242.66, -7.5) mm, rotated rx 180 ry 0 rz -180 deg; joints [-9.087, -42.042, 105.492, 169.863, 63.809, -175.488]
  MoveL 3215 to (307.88, 246.32, -7.5) mm, rotated rx 180 ry 0 rz -180 deg; joints [-9.219, -42.02, 105.429, 169.712, 63.778, -175.415]
  MoveL 3216 to (308, 250, -7.5) mm, rotated rx -180 ry 0 rz -180 deg; joints [-9.354, -42.004, 105.38, 169.56, 63.758, -175.342]
  MoveL 3217 to (296, 250, -7.5) mm, rotated rx -180 ry 0 rz 180 deg; joints [-9.427, -42.278, 106.184, 169.525, 64.284, -175.414]
  MoveL 3218 to (295.91, 252.92, -7.5) mm, rotated rx -180 ry 0 rz -180 deg; joints [-9.536, -42.269, 106.158, 169.404, 64.276, -175.358]
  MoveL 3219 to (295.63, 255.82, -7.5) mm, rotated rx 180 ry 0 rz -180 deg; joints [-9.645, -42.264, 106.144, 169.282, 64.276, -175.303]
  MoveL 3220 to (295.17, 258.71, -7.5) mm, rotated rx -180 ry 0 rz -180 deg; joints [-9.755, -42.264, 106.141, 169.161, 64.283, -175.251]
  MoveL 3221 to (294.53, 261.55, -7.5) mm, rotated rx -180 ry 0 rz -180 deg; joints [-9.864, -42.267, 106.152, 169.04, 64.299, -175.2]
  MoveL 3222 to (293.7, 264.35, -7.5) mm, rotated rx -180 ry 0 rz -180 deg; joints [-9.973, -42.275, 106.174, 168.921, 64.322, -175.15]
  MoveL 3223 to (292.7, 267.1, -7.5) mm, rotated rx 180 ry 0 rz -180 deg; joints [-10.081, -42.286, 106.208, 168.804, 64.354, -175.104]
  MoveL 3224 to (291.53, 269.77, -7.5) mm, rotated rx 180 ry 0 rz -180 deg; joints [-10.187, -42.302, 106.254, 168.689, 64.393, -175.059]
  MoveL 3225 to (290.2, 272.37, -7.5) mm, rotated rx 180 ry 0 rz -180 deg; joints [-10.292, -42.321, 106.312, 168.577, 64.439, -175.018]
  MoveL 3226 to (288.7, 274.87, -7.5) mm, rotated rx -180 ry 0 rz -180 deg; joints [-10.395, -42.345, 106.381, 168.468, 64.493, -174.979]
  MoveL 3227 to (287.04, 277.27, -7.5) mm, rotated rx 180 ry 0 rz 180 deg; joints [-10.495, -42.372, 106.462, 168.362, 64.554, -174.943]
  MoveL 3228 to (285.24, 279.57, -7.5) mm, rotated rx 180 ry 0 rz 180 deg; joints [-10.593, -42.403, 106.553, 168.261, 64.622, -174.911]
  MoveL 3229 to (283.29, 281.74, -7.5) mm, rotated rx 180 ry 0 rz 180 deg; joints [-10.687, -42.438, 106.655, 168.164, 64.697, -174.882]
  MoveL 3230 to (281.21, 283.79, -7.5) mm, rotated rx 180 ry 0 rz 180 deg; joints [-10.777, -42.475, 106.768, 168.071, 64.778, -174.856]
  MoveL 3231 to (279.01, 285.7, -7.5) mm, rotated rx -180 ry 0 rz -180 deg; joints [-10.864, -42.516, 106.89, 167.984, 64.865, -174.834]
  MoveL 3232 to (276.68, 287.47, -7.5) mm, rotated rx 180 ry 0 rz -180 deg; joints [-10.946, -42.561, 107.021, 167.902, 64.957, -174.816]
  MoveL 3233 to (274.25, 289.09, -7.5) mm, rotated rx -180 ry 0 rz -180 deg; joints [-11.024, -42.607, 107.161, 167.826, 65.055, -174.801]
  MoveL 3234 to (271.72, 290.55, -7.5) mm, rotated rx -180 ry 0 rz 180 deg; joints [-11.096, -42.657, 107.309, 167.755, 65.158, -174.791]
  MoveL 3235 to (269.11, 291.84, -7.5) mm, rotated rx 180 ry 0 rz 180 deg; joints [-11.164, -42.709, 107.464, 167.692, 65.266, -174.784]
  MoveL 3236 to (266.42, 292.97, -7.5) mm, rotated rx 180 ry 0 rz 180 deg; joints [-11.226, -42.763, 107.627, 167.634, 65.377, -174.781]
  MoveL 3237 to (263.66, 293.93, -7.5) mm, rotated rx -180 ry 0 rz -180 deg; joints [-11.282, -42.819, 107.796, 167.584, 65.492, -174.782]
  MoveL 3238 to (260.84, 294.7, -7.5) mm, rotated rx 180 ry 0 rz -180 deg; joints [-11.332, -42.877, 107.97, 167.54, 65.611, -174.787]
  MoveL 3239 to (257.99, 295.3, -7.5) mm, rotated rx 180 ry 0 rz 180 deg; joints [-11.376, -42.936, 108.15, 167.504, 65.732, -174.796]
  MoveL 3240 to (255.1, 295.72, -7.5) mm, rotated rx -180 ry 0 rz -180 deg; joints [-11.414, -42.997, 108.334, 167.475, 65.856, -174.808]
  MoveL 3241 to (252.19, 295.95, -7.5) mm, rotated rx 180 ry 0 rz -180 deg; joints [-11.444, -43.058, 108.521, 167.454, 65.982, -174.824]
  MoveL 3242 to (249.27, 295.99, -7.5) mm, rotated rx 180 ry 0 rz 180 deg; joints [-11.468, -43.12, 108.711, 167.44, 66.109, -174.844]
  MoveL 3243 to (246.35, 295.86, -7.5) mm, rotated rx 180 ry 0 rz -180 deg; joints [-11.486, -43.183, 108.903, 167.434, 66.236, -174.867]
  MoveL 3244 to (243.45, 295.53, -7.5) mm, rotated rx -180 ry 0 rz -180 deg; joints [-11.496, -43.246, 109.096, 167.435, 66.365, -174.894]
  MoveL 3245 to (240.58, 295.02, -7.5) mm, rotated rx 180 ry 0 rz -180 deg; joints [-11.499, -43.309, 109.29, 167.445, 66.493, -174.924]
  MoveL 3246 to (237.74, 294.34, -7.5) mm, rotated rx 180 ry 0 rz 180 deg; joints [-11.494, -43.371, 109.484, 167.461, 66.62, -174.956]
  MoveL 3247 to (234.95, 293.47, -7.5) mm, rotated rx -180 ry 0 rz -180 deg; joints [-11.483, -43.433, 109.676, 167.486, 66.746, -174.992]
  MoveL 3248 to (232.23, 292.43, -7.5) mm, rotated rx -180 ry 0 rz -180 deg; joints [-11.464, -43.495, 109.867, 167.518, 66.871, -175.031]
  MoveL 3249 to (229.57, 291.22, -7.5) mm, rotated rx 180 ry 0 rz 180 deg; joints [-11.439, -43.555, 110.054, 167.558, 66.993, -175.071]
  MoveL 3250 to (227, 289.84, -7.5) mm, rotated rx 180 ry 0 rz -180 deg; joints [-11.406, -43.614, 110.239, 167.605, 67.113, -175.115]
  MoveL 3251 to (224.52, 288.3, -7.5) mm, rotated rx 180 ry 0 rz -180 deg; joints [-11.366, -43.671, 110.419, 167.659, 67.23, -175.16]
  MoveL 3252 to (222.14, 286.61, -7.5) mm, rotated rx 180 ry 0 rz -180 deg; joints [-11.319, -43.727, 110.595, 167.72, 67.343, -175.207]
  MoveL 3253 to (219.88, 284.76, -7.5) mm, rotated rx 180 ry 0 rz -180 deg; joints [-11.266, -43.78, 110.765, 167.788, 67.452, -175.256]
  MoveL 3254 to (217.73, 282.78, -7.5) mm, rotated rx 180 ry 0 rz 180 deg; joints [-11.206, -43.832, 110.928, 167.863, 67.557, -175.306]
  MoveL 3255 to (215.72, 280.67, -7.5) mm, rotated rx -180 ry 0 rz -180 deg; joints [-11.139, -43.881, 111.085, 167.943, 67.657, -175.358]
  MoveL 3256 to (213.84, 278.44, -7.5) mm, rotated rx -180 ry 0 rz 180 deg; joints [-11.067, -43.928, 111.234, 168.03, 67.751, -175.411]
  MoveL 3257 to (212.11, 276.08, -7.5) mm, rotated rx 180 ry 0 rz -180 deg; joints [-10.989, -43.972, 111.375, 168.122, 67.839, -175.464]
  MoveL 3258 to (210.53, 273.63, -7.5) mm, rotated rx 180 ry 0 rz 180 deg; joints [-10.905, -44.013, 111.507, 168.22, 67.922, -175.518]
  MoveL 3259 to (209.11, 271.08, -7.5) mm, rotated rx -180 ry 0 rz -180 deg; joints [-10.817, -44.051, 111.629, 168.322, 67.998, -175.572]
  MoveL 3260 to (207.86, 268.44, -7.5) mm, rotated rx -180 ry 0 rz -180 deg; joints [-10.723, -44.086, 111.742, 168.429, 68.067, -175.627]
  MoveL 3261 to (206.77, 265.73, -7.5) mm, rotated rx 180 ry 0 rz 180 deg; joints [-10.625, -44.118, 111.845, 168.54, 68.129, -175.681]
  MoveL 3262 to (205.86, 262.96, -7.5) mm, rotated rx 180 ry 0 rz -180 deg; joints [-10.523, -44.146, 111.936, 168.654, 68.183, -175.735]
  MoveL 3263 to (205.13, 260.13, -7.5) mm, rotated rx -180 ry 0 rz 180 deg; joints [-10.418, -44.171, 112.017, 168.772, 68.23, -175.789]
  MoveL 3264 to (204.58, 257.27, -7.5) mm, rotated rx 180 ry 0 rz 180 deg; joints [-10.31, -44.192, 112.086, 168.892, 68.269, -175.842]
  MoveL 3265 to (204.21, 254.37, -7.5) mm, rotated rx -180 ry 0 rz 180 deg; joints [-10.199, -44.21, 112.143, 169.014, 68.3, -175.894]
  MoveL 3266 to (204.02, 251.46, -7.5) mm, rotated rx -180 ry 0 rz -180 deg; joints [-10.086, -44.224, 112.189, 169.138, 68.323, -175.946]
  MoveL 3267 to (204.02, 248.54, -7.5) mm, rotated rx -180 ry 0 rz -180 deg; joints [-9.971, -44.234, 112.222, 169.263, 68.337, -175.996]
  MoveL 3268 to (204.21, 245.63, -7.5) mm, rotated rx -180 ry 0 rz -180 deg; joints [-9.855, -44.24, 112.243, 169.388, 68.343, -176.045]
  MoveL 3269 to (204.58, 242.73, -7.5) mm, rotated rx -180 ry 0 rz 180 deg; joints [-9.739, -44.243, 112.251, 169.513, 68.341, -176.092]
  MoveL 3270 to (205.13, 239.87, -7.5) mm, rotated rx 180 ry 0 rz -180 deg; joints [-9.622, -44.242, 112.247, 169.638, 68.33, -176.137]
  MoveL 3271 to (205.86, 237.04, -7.5) mm, rotated rx -180 ry 0 rz -180 deg; joints [-9.506, -44.237, 112.23, 169.762, 68.311, -176.181]
  MoveL 3272 to (206.77, 234.27, -7.5) mm, rotated rx 180 ry 0 rz -180 deg; joints [-9.391, -44.228, 112.202, 169.884, 68.284, -176.223]
  MoveL 3273 to (207.86, 231.56, -7.5) mm, rotated rx 180 ry 0 rz 180 deg; joints [-9.277, -44.215, 112.16, 170.005, 68.249, -176.263]
  MoveL 3274 to (209.11, 228.92, -7.5) mm, rotated rx 180 ry 0 rz 180 deg; joints [-9.166, -44.199, 112.107, 170.122, 68.205, -176.301]
  MoveL 3275 to (210.53, 226.37, -7.5) mm, rotated rx -180 ry 0 rz 180 deg; joints [-9.056, -44.179, 112.042, 170.237, 68.154, -176.336]
  MoveL 3276 to (212.11, 223.92, -7.5) mm, rotated rx -180 ry 0 rz -180 deg; joints [-8.95, -44.155, 111.966, 170.347, 68.095, -176.369]
  MoveL 3277 to (213.84, 221.56, -7.5) mm, rotated rx 180 ry 0 rz 180 deg; joints [-8.847, -44.128, 111.878, 170.454, 68.028, -176.4]
  MoveL 3278 to (215.72, 219.33, -7.5) mm, rotated rx 180 ry 0 rz 180 deg; joints [-8.747, -44.097, 111.779, 170.556, 67.955, -176.428]
  MoveL 3279 to (217.73, 217.22, -7.5) mm, rotated rx -180 ry 0 rz 180 deg; joints [-8.652, -44.064, 111.67, 170.654, 67.874, -176.453]
  MoveL 3280 to (219.88, 215.24, -7.5) mm, rotated rx 180 ry 0 rz 180 deg; joints [-8.562, -44.027, 111.55, 170.746, 67.788, -176.475]
  MoveL 3281 to (222.14, 213.4, -7.5) mm, rotated rx -180 ry 0 rz -180 deg; joints [-8.477, -43.986, 111.421, 170.832, 67.695, -176.495]
  MoveL 3282 to (224.52, 211.7, -7.5) mm, rotated rx 180 ry 0 rz 180 deg; joints [-8.397, -43.943, 111.284, 170.912, 67.596, -176.511]
  MoveL 3283 to (227, 210.16, -7.5) mm, rotated rx -180 ry 0 rz 180 deg; joints [-8.322, -43.898, 111.137, 170.986, 67.493, -176.525]
  MoveL 3284 to (229.57, 208.78, -7.5) mm, rotated rx -180 ry 0 rz -180 deg; joints [-8.254, -43.849, 110.983, 171.053, 67.384, -176.535]
  MoveL 3285 to (232.23, 207.57, -7.5) mm, rotated rx 180 ry 0 rz -180 deg; joints [-8.192, -43.799, 110.822, 171.113, 67.271, -176.543]
  MoveL 3286 to (234.95, 206.53, -7.5) mm, rotated rx -180 ry 0 rz -180 deg; joints [-8.136, -43.746, 110.654, 171.166, 67.154, -176.547]
  MoveL 3287 to (237.74, 205.66, -7.5) mm, rotated rx 180 ry 0 rz 180 deg; joints [-8.087, -43.691, 110.48, 171.212, 67.034, -176.548]
  MoveL 3288 to (240.58, 204.98, -7.5) mm, rotated rx 180 ry 0 rz 180 deg; joints [-8.045, -43.634, 110.302, 171.25, 66.911, -176.546]
  MoveL 3289 to (243.45, 204.47, -7.5) mm, rotated rx -180 ry 0 rz -180 deg; joints [-8.009, -43.575, 110.119, 171.28, 66.786, -176.54]
  MoveL 3290 to (246.35, 204.14, -7.5) mm, rotated rx 180 ry 0 rz 180 deg; joints [-7.981, -43.516, 109.932, 171.302, 66.658, -176.531]
  MoveL 3291 to (249.27, 204.01, -7.5) mm, rotated rx -180 ry 0 rz -180 deg; joints [-7.96, -43.455, 109.742, 171.317, 66.53, -176.519]
  MoveL 3292 to (252.19, 204.05, -7.5) mm, rotated rx -180 ry 0 rz -180 deg; joints [-7.946, -43.393, 109.55, 171.323, 66.4, -176.504]
  MoveL 3293 to (255.1, 204.28, -7.5) mm, rotated rx 180 ry 0 rz -180 deg; joints [-7.939, -43.331, 109.357, 171.322, 66.27, -176.485]
  MoveL 3294 to (257.99, 204.7, -7.5) mm, rotated rx -180 ry 0 rz 180 deg; joints [-7.94, -43.268, 109.163, 171.313, 66.141, -176.463]
  MoveL 3295 to (260.84, 205.3, -7.5) mm, rotated rx -180 ry 0 rz 180 deg; joints [-7.947, -43.205, 108.97, 171.296, 66.012, -176.438]
  MoveL 3296 to (263.66, 206.07, -7.5) mm, rotated rx -180 ry 0 rz 180 deg; joints [-7.962, -43.142, 108.777, 171.271, 65.885, -176.41]
  MoveL 3297 to (266.42, 207.03, -7.5) mm, rotated rx -180 ry 0 rz -180 deg; joints [-7.984, -43.08, 108.586, 171.238, 65.759, -176.379]
  MoveL 3298 to (269.11, 208.16, -7.5) mm, rotated rx -180 ry 0 rz -180 deg; joints [-8.012, -43.018, 108.398, 171.198, 65.636, -176.345]
  MoveL 3299 to (271.72, 209.45, -7.5) mm, rotated rx 180 ry 0 rz 180 deg; joints [-8.047, -42.957, 108.213, 171.151, 65.516, -176.308]
  MoveL 3300 to (274.25, 210.91, -7.5) mm, rotated rx -180 ry 0 rz 180 deg; joints [-8.089, -42.897, 108.032, 171.097, 65.398, -176.269]
  MoveL 3301 to (276.68, 212.53, -7.5) mm, rotated rx -180 ry 0 rz -180 deg; joints [-8.137, -42.839, 107.855, 171.036, 65.285, -176.227]
  MoveL 3302 to (279.01, 214.3, -7.5) mm, rotated rx 180 ry 0 rz 180 deg; joints [-8.191, -42.782, 107.684, 170.968, 65.176, -176.182]
  MoveL 3303 to (281.21, 216.21, -7.5) mm, rotated rx 180 ry 0 rz 180 deg; joints [-8.251, -42.727, 107.52, 170.894, 65.071, -176.135]
  MoveL 3304 to (283.29, 218.26, -7.5) mm, rotated rx -180 ry 0 rz -180 deg; joints [-8.317, -42.675, 107.362, 170.814, 64.972, -176.086]
  MoveL 3305 to (285.24, 220.43, -7.5) mm, rotated rx -180 ry 0 rz 180 deg; joints [-8.388, -42.624, 107.211, 170.728, 64.877, -176.035]
  MoveL 3306 to (287.04, 222.73, -7.5) mm, rotated rx 180 ry 0 rz 180 deg; joints [-8.464, -42.576, 107.068, 170.637, 64.789, -175.983]
  MoveL 3307 to (288.7, 225.13, -7.5) mm, rotated rx -180 ry 0 rz 180 deg; joints [-8.545, -42.531, 106.934, 170.541, 64.707, -175.929]
  MoveL 3308 to (290.2, 227.64, -7.5) mm, rotated rx 180 ry 0 rz 180 deg; joints [-8.63, -42.489, 106.809, 170.441, 64.631, -175.873]
  MoveL 3309 to (291.53, 230.23, -7.5) mm, rotated rx 180 ry 0 rz 180 deg; joints [-8.719, -42.45, 106.693, 170.336, 64.562, -175.817]
  MoveL 3310 to (292.7, 232.9, -7.5) mm, rotated rx 180 ry 0 rz 180 deg; joints [-8.812, -42.415, 106.587, 170.228, 64.5, -175.76]
  MoveL 3311 to (293.7, 235.65, -7.5) mm, rotated rx 180 ry 0 rz 180 deg; joints [-8.908, -42.383, 106.492, 170.117, 64.445, -175.702]
  MoveL 3312 to (294.53, 238.45, -7.5) mm, rotated rx -180 ry 0 rz 180 deg; joints [-9.007, -42.354, 106.408, 170.002, 64.397, -175.644]
  MoveL 3313 to (295.17, 241.29, -7.5) mm, rotated rx -180 ry 0 rz -180 deg; joints [-9.109, -42.329, 106.335, 169.885, 64.357, -175.586]
  MoveL 3314 to (295.63, 244.18, -7.5) mm, rotated rx -180 ry 0 rz -180 deg; joints [-9.214, -42.308, 106.273, 169.767, 64.325, -175.528]
  MoveL 3315 to (295.91, 247.08, -7.5) mm, rotated rx -180 ry 0 rz -180 deg; joints [-9.32, -42.291, 106.223, 169.647, 64.301, -175.47]
  MoveL 3316 to (296, 250, -7.5) mm, rotated rx -180 ry 0 rz 180 deg; joints [-9.427, -42.278, 106.184, 169.525, 64.284, -175.414]
  MoveL 3317 to (284, 250, -7.5) mm, rotated rx 180 ry 0 rz -180 deg; joints [-9.502, -42.548, 106.984, 169.489, 64.811, -175.485]
  MoveL 3318 to (283.93, 252.16, -7.5) mm, rotated rx -180 ry 0 rz 180 deg; joints [-9.582, -42.542, 106.964, 169.399, 64.805, -175.445]
  MoveL 3319 to (283.73, 254.3, -7.5) mm, rotated rx 180 ry 0 rz -180 deg; joints [-9.664, -42.538, 106.954, 169.309, 64.804, -175.405]
  MoveL 3320 to (283.39, 256.43, -7.5) mm, rotated rx 180 ry 0 rz 180 deg; joints [-9.745, -42.537, 106.952, 169.219, 64.81, -175.366]
  MoveL 3321 to (282.91, 258.54, -7.5) mm, rotated rx -180 ry 0 rz -180 deg; joints [-9.827, -42.54, 106.959, 169.129, 64.821, -175.329]
  MoveL 3322 to (282.3, 260.61, -7.5) mm, rotated rx -180 ry 0 rz -180 deg; joints [-9.908, -42.545, 106.976, 169.041, 64.839, -175.294]
  MoveL 3323 to (281.56, 262.64, -7.5) mm, rotated rx -180 ry 0 rz 180 deg; joints [-9.988, -42.554, 107.001, 168.954, 64.862, -175.26]
  MoveL 3324 to (280.7, 264.61, -7.5) mm, rotated rx -180 ry 0 rz -180 deg; joints [-10.068, -42.565, 107.035, 168.869, 64.891, -175.227]
  MoveL 3325 to (279.71, 266.53, -7.5) mm, rotated rx 180 ry 0 rz 180 deg; joints [-10.146, -42.58, 107.078, 168.786, 64.925, -175.197]
  MoveL 3326 to (278.6, 268.38, -7.5) mm, rotated rx -180 ry 0 rz 180 deg; joints [-10.222, -42.597, 107.13, 168.705, 64.965, -175.169]
  MoveL 3327 to (277.38, 270.16, -7.5) mm, rotated rx -180 ry 0 rz 180 deg; joints [-10.297, -42.617, 107.189, 168.626, 65.01, -175.143]
  MoveL 3328 to (276.05, 271.85, -7.5) mm, rotated rx -180 ry 0 rz -180 deg; joints [-10.369, -42.64, 107.257, 168.551, 65.061, -175.119]
  MoveL 3329 to (274.61, 273.46, -7.5) mm, rotated rx 180 ry 0 rz -180 deg; joints [-10.439, -42.665, 107.333, 168.479, 65.116, -175.098]
  MoveL 3330 to (273.07, 274.98, -7.5) mm, rotated rx -180 ry 0 rz -180 deg; joints [-10.506, -42.693, 107.416, 168.41, 65.176, -175.079]
  MoveL 3331 to (271.44, 276.39, -7.5) mm, rotated rx -180 ry 0 rz 180 deg; joints [-10.57, -42.723, 107.506, 168.346, 65.24, -175.063]
  MoveL 3332 to (269.72, 277.7, -7.5) mm, rotated rx 180 ry 0 rz -180 deg; joints [-10.631, -42.755, 107.603, 168.285, 65.309, -175.049]
  MoveL 3333 to (267.93, 278.89, -7.5) mm, rotated rx 180 ry 0 rz 180 deg; joints [-10.688, -42.79, 107.707, 168.228, 65.382, -175.039]
  MoveL 3334 to (266.06, 279.97, -7.5) mm, rotated rx -180 ry 0 rz -180 deg; joints [-10.742, -42.826, 107.817, 168.176, 65.458, -175.031]
  MoveL 3335 to (264.12, 280.93, -7.5) mm, rotated rx -180 ry 0 rz -180 deg; joints [-10.792, -42.864, 107.932, 168.129, 65.538, -175.025]
  MoveL 3336 to (262.13, 281.76, -7.5) mm, rotated rx -180 ry 0 rz -180 deg; joints [-10.837, -42.904, 108.052, 168.087, 65.621, -175.023]
  MoveL 3337 to (260.1, 282.47, -7.5) mm, rotated rx -180 ry 0 rz -180 deg; joints [-10.879, -42.945, 108.177, 168.05, 65.706, -175.023]
  MoveL 3338 to (258.02, 283.04, -7.5) mm, rotated rx 180 ry 0 rz 180 deg; joints [-10.915, -42.988, 108.306, 168.018, 65.794, -175.027]
  MoveL 3339 to (255.9, 283.48, -7.5) mm, rotated rx -180 ry 0 rz 180 deg; joints [-10.947, -43.031, 108.439, 167.991, 65.884, -175.033]
  MoveL 3340 to (253.77, 283.79, -7.5) mm, rotated rx -180 ry 0 rz -180 deg; joints [-10.974, -43.076, 108.575, 167.97, 65.976, -175.041]
  MoveL 3341 to (251.62, 283.96, -7.5) mm, rotated rx -180 ry 0 rz -180 deg; joints [-10.997, -43.121, 108.714, 167.954, 66.069, -175.053]
  MoveL 3342 to (249.46, 284, -7.5) mm, rotated rx -180 ry 0 rz -180 deg; joints [-11.014, -43.167, 108.854, 167.944, 66.163, -175.067]
  MoveL 3343 to (247.31, 283.89, -7.5) mm, rotated rx 180 ry 0 rz -180 deg; joints [-11.026, -43.214, 108.996, 167.94, 66.258, -175.083]
  MoveL 3344 to (245.16, 283.65, -7.5) mm, rotated rx 180 ry 0 rz 180 deg; joints [-11.033, -43.26, 109.139, 167.942, 66.352, -175.103]
  MoveL 3345 to (243.04, 283.28, -7.5) mm, rotated rx 180 ry 0 rz 180 deg; joints [-11.034, -43.306, 109.282, 167.949, 66.447, -175.124]
  MoveL 3346 to (240.94, 282.77, -7.5) mm, rotated rx 180 ry 0 rz -180 deg; joints [-11.03, -43.353, 109.425, 167.962, 66.542, -175.148]
  MoveL 3347 to (238.88, 282.13, -7.5) mm, rotated rx 180 ry 0 rz -180 deg; joints [-11.021, -43.399, 109.568, 167.98, 66.635, -175.173]
  MoveL 3348 to (236.86, 281.36, -7.5) mm, rotated rx -180 ry 0 rz -180 deg; joints [-11.007, -43.444, 109.708, 168.004, 66.727, -175.201]
  MoveL 3349 to (234.9, 280.46, -7.5) mm, rotated rx 180 ry 0 rz -180 deg; joints [-10.987, -43.488, 109.847, 168.034, 66.818, -175.231]
  MoveL 3350 to (233, 279.44, -7.5) mm, rotated rx 180 ry 0 rz -180 deg; joints [-10.962, -43.532, 109.983, 168.069, 66.906, -175.262]
  MoveL 3351 to (231.17, 278.31, -7.5) mm, rotated rx -180 ry 0 rz -180 deg; joints [-10.932, -43.575, 110.117, 168.11, 66.992, -175.295]
  MoveL 3352 to (229.41, 277.06, -7.5) mm, rotated rx 180 ry 0 rz 180 deg; joints [-10.897, -43.616, 110.246, 168.155, 67.076, -175.33]
  MoveL 3353 to (227.73, 275.7, -7.5) mm, rotated rx -180 ry 0 rz 180 deg; joints [-10.857, -43.656, 110.371, 168.206, 67.156, -175.366]
  MoveL 3354 to (226.15, 274.23, -7.5) mm, rotated rx 180 ry 0 rz -180 deg; joints [-10.813, -43.694, 110.492, 168.261, 67.233, -175.403]
  MoveL 3355 to (224.66, 272.67, -7.5) mm, rotated rx -180 ry 0 rz -180 deg; joints [-10.763, -43.731, 110.608, 168.321, 67.307, -175.441]
  MoveL 3356 to (223.27, 271.02, -7.5) mm, rotated rx 180 ry 0 rz 180 deg; joints [-10.71, -43.766, 110.718, 168.385, 67.376, -175.479]
  MoveL 3357 to (222, 269.28, -7.5) mm, rotated rx -180 ry 0 rz -180 deg; joints [-10.652, -43.798, 110.821, 168.454, 67.441, -175.519]
  MoveL 3358 to (220.83, 267.47, -7.5) mm, rotated rx 180 ry 0 rz 180 deg; joints [-10.59, -43.829, 110.919, 168.526, 67.502, -175.559]
  MoveL 3359 to (219.78, 265.58, -7.5) mm, rotated rx -180 ry 0 rz 180 deg; joints [-10.525, -43.857, 111.009, 168.602, 67.557, -175.599]
  MoveL 3360 to (218.85, 263.63, -7.5) mm, rotated rx 180 ry 0 rz 180 deg; joints [-10.456, -43.884, 111.092, 168.681, 67.608, -175.639]
  MoveL 3361 to (218.05, 261.63, -7.5) mm, rotated rx -180 ry 0 rz -180 deg; joints [-10.384, -43.907, 111.168, 168.762, 67.653, -175.68]
  MoveL 3362 to (217.38, 259.58, -7.5) mm, rotated rx 180 ry 0 rz 180 deg; joints [-10.309, -43.928, 111.235, 168.847, 67.693, -175.72]
  MoveL 3363 to (216.84, 257.49, -7.5) mm, rotated rx 180 ry 0 rz 180 deg; joints [-10.232, -43.947, 111.295, 168.933, 67.728, -175.76]
  MoveL 3364 to (216.43, 255.37, -7.5) mm, rotated rx 180 ry 0 rz 180 deg; joints [-10.152, -43.963, 111.346, 169.022, 67.756, -175.8]
  MoveL 3365 to (216.15, 253.23, -7.5) mm, rotated rx -180 ry 0 rz 180 deg; joints [-10.071, -43.976, 111.388, 169.112, 67.779, -175.839]
  MoveL 3366 to (216.02, 251.08, -7.5) mm, rotated rx -180 ry 0 rz -180 deg; joints [-9.988, -43.986, 111.421, 169.203, 67.795, -175.878]
  MoveL 3367 to (216.02, 248.92, -7.5) mm, rotated rx 180 ry 0 rz 180 deg; joints [-9.904, -43.994, 111.446, 169.295, 67.806, -175.915]
  MoveL 3368 to (216.15, 246.77, -7.5) mm, rotated rx 180 ry 0 rz -180 deg; joints [-9.819, -43.999, 111.461, 169.387, 67.81, -175.952]
  MoveL 3369 to (216.43, 244.63, -7.5) mm, rotated rx 180 ry 0 rz 180 deg; joints [-9.733, -44.001, 111.467, 169.479, 67.808, -175.988]
  MoveL 3370 to (216.84, 242.51, -7.5) mm, rotated rx -180 ry 0 rz -180 deg; joints [-9.648, -44, 111.464, 169.571, 67.8, -176.022]
  MoveL 3371 to (217.38, 240.42, -7.5) mm, rotated rx 180 ry 0 rz 180 deg; joints [-9.563, -43.996, 111.452, 169.662, 67.786, -176.055]
  MoveL 3372 to (218.05, 238.37, -7.5) mm, rotated rx -180 ry 0 rz 180 deg; joints [-9.478, -43.989, 111.431, 169.752, 67.766, -176.087]
  MoveL 3373 to (218.85, 236.37, -7.5) mm, rotated rx -180 ry 0 rz -180 deg; joints [-9.395, -43.98, 111.401, 169.841, 67.74, -176.117]
  MoveL 3374 to (219.78, 234.42, -7.5) mm, rotated rx 180 ry 0 rz 180 deg; joints [-9.313, -43.968, 111.361, 169.927, 67.708, -176.145]
  MoveL 3375 to (220.83, 232.54, -7.5) mm, rotated rx 180 ry 0 rz -180 deg; joints [-9.233, -43.953, 111.313, 170.011, 67.67, -176.172]
  MoveL 3376 to (221.99, 230.72, -7.5) mm, rotated rx 180 ry 0 rz 180 deg; joints [-9.155, -43.935, 111.257, 170.093, 67.626, -176.196]
  MoveL 3377 to (223.27, 228.98, -7.5) mm, rotated rx 180 ry 0 rz 180 deg; joints [-9.079, -43.915, 111.192, 170.172, 67.578, -176.219]
  MoveL 3378 to (224.66, 227.33, -7.5) mm, rotated rx 180 ry 0 rz 180 deg; joints [-9.006, -43.892, 111.119, 170.247, 67.524, -176.24]
  MoveL 3379 to (226.15, 225.77, -7.5) mm, rotated rx 180 ry 0 rz 180 deg; joints [-8.936, -43.867, 111.039, 170.319, 67.464, -176.259]
  MoveL 3380 to (227.73, 224.3, -7.5) mm, rotated rx -180 ry 0 rz 180 deg; joints [-8.869, -43.839, 110.951, 170.386, 67.401, -176.276]
  MoveL 3381 to (229.41, 222.94, -7.5) mm, rotated rx -180 ry 0 rz -180 deg; joints [-8.806, -43.809, 110.856, 170.45, 67.332, -176.29]
  MoveL 3382 to (231.17, 221.69, -7.5) mm, rotated rx -180 ry 0 rz -180 deg; joints [-8.747, -43.777, 110.754, 170.509, 67.26, -176.303]
  MoveL 3383 to (233, 220.56, -7.5) mm, rotated rx 180 ry 0 rz -180 deg; joints [-8.692, -43.743, 110.646, 170.564, 67.184, -176.312]
  MoveL 3384 to (234.9, 219.54, -7.5) mm, rotated rx 180 ry 0 rz -180 deg; joints [-8.641, -43.707, 110.533, 170.613, 67.104, -176.32]
  MoveL 3385 to (236.86, 218.64, -7.5) mm, rotated rx 180 ry 0 rz -180 deg; joints [-8.595, -43.669, 110.414, 170.658, 67.021, -176.325]
  MoveL 3386 to (238.88, 217.87, -7.5) mm, rotated rx -180 ry 0 rz -180 deg; joints [-8.553, -43.63, 110.29, 170.697, 66.935, -176.328]
  MoveL 3387 to (240.94, 217.23, -7.5) mm, rotated rx -180 ry 0 rz -180 deg; joints [-8.517, -43.589, 110.162, 170.731, 66.846, -176.328]
  MoveL 3388 to (243.04, 216.72, -7.5) mm, rotated rx -180 ry 0 rz -180 deg; joints [-8.485, -43.547, 110.03, 170.759, 66.755, -176.326]
  MoveL 3389 to (245.16, 216.35, -7.5) mm, rotated rx 180 ry 0 rz 180 deg; joints [-8.458, -43.504, 109.894, 170.782, 66.663, -176.322]
  MoveL 3390 to (247.31, 216.11, -7.5) mm, rotated rx -180 ry 0 rz -180 deg; joints [-8.437, -43.459, 109.757, 170.799, 66.569, -176.314]
  MoveL 3391 to (249.46, 216, -7.5) mm, rotated rx -180 ry 0 rz -180 deg; joints [-8.421, -43.414, 109.616, 170.81, 66.474, -176.305]
  MoveL 3392 to (251.62, 216.04, -7.5) mm, rotated rx 180 ry 0 rz 180 deg; joints [-8.41, -43.369, 109.475, 170.815, 66.379, -176.293]
  MoveL 3393 to (253.77, 216.21, -7.5) mm, rotated rx -180 ry 0 rz 180 deg; joints [-8.404, -43.322, 109.332, 170.814, 66.283, -176.279]
  MoveL 3394 to (255.9, 216.52, -7.5) mm, rotated rx 180 ry 0 rz -180 deg; joints [-8.404, -43.276, 109.189, 170.808, 66.187, -176.262]
  MoveL 3395 to (258.02, 216.96, -7.5) mm, rotated rx -180 ry 0 rz -180 deg; joints [-8.409, -43.23, 109.046, 170.796, 66.092, -176.243]
  MoveL 3396 to (260.1, 217.53, -7.5) mm, rotated rx -180 ry 0 rz 180 deg; joints [-8.419, -43.183, 108.903, 170.778, 65.998, -176.221]
  MoveL 3397 to (262.13, 218.24, -7.5) mm, rotated rx 180 ry 0 rz 180 deg; joints [-8.434, -43.137, 108.762, 170.754, 65.905, -176.198]
  MoveL 3398 to (264.12, 219.07, -7.5) mm, rotated rx 180 ry 0 rz -180 deg; joints [-8.455, -43.092, 108.623, 170.725, 65.814, -176.172]
  MoveL 3399 to (266.06, 220.03, -7.5) mm, rotated rx 180 ry 0 rz 180 deg; joints [-8.48, -43.047, 108.486, 170.69, 65.725, -176.144]
  MoveL 3400 to (267.93, 221.11, -7.5) mm, rotated rx -180 ry 0 rz -180 deg; joints [-8.51, -43.003, 108.352, 170.651, 65.638, -176.115]
  MoveL 3401 to (269.72, 222.3, -7.5) mm, rotated rx 180 ry 0 rz 180 deg; joints [-8.546, -42.96, 108.221, 170.606, 65.554, -176.083]
  MoveL 3402 to (271.44, 223.61, -7.5) mm, rotated rx -180 ry 0 rz -180 deg; joints [-8.585, -42.918, 108.095, 170.556, 65.473, -176.05]
  MoveL 3403 to (273.07, 225.02, -7.5) mm, rotated rx 180 ry 0 rz 180 deg; joints [-8.629, -42.878, 107.973, 170.501, 65.396, -176.015]
  MoveL 3404 to (274.61, 226.54, -7.5) mm, rotated rx 180 ry 0 rz -180 deg; joints [-8.678, -42.839, 107.856, 170.442, 65.322, -175.979]
  MoveL 3405 to (276.05, 228.15, -7.5) mm, rotated rx -180 ry 0 rz 180 deg; joints [-8.73, -42.802, 107.744, 170.379, 65.252, -175.941]
  MoveL 3406 to (277.38, 229.84, -7.5) mm, rotated rx -180 ry 0 rz -180 deg; joints [-8.786, -42.767, 107.638, 170.312, 65.187, -175.902]
  MoveL 3407 to (278.6, 231.62, -7.5) mm, rotated rx -180 ry 0 rz 180 deg; joints [-8.846, -42.734, 107.539, 170.241, 65.125, -175.862]
  MoveL 3408 to (279.71, 233.47, -7.5) mm, rotated rx -180 ry 0 rz -180 deg; joints [-8.909, -42.703, 107.446, 170.167, 65.069, -175.821]
  MoveL 3409 to (280.7, 235.39, -7.5) mm, rotated rx 180 ry 0 rz 180 deg; joints [-8.975, -42.674, 107.361, 170.09, 65.018, -175.78]
  MoveL 3410 to (281.56, 237.36, -7.5) mm, rotated rx -180 ry 0 rz -180 deg; joints [-9.044, -42.648, 107.282, 170.01, 64.972, -175.738]
  MoveL 3411 to (282.3, 239.39, -7.5) mm, rotated rx 180 ry 0 rz 180 deg; joints [-9.115, -42.625, 107.212, 169.927, 64.931, -175.696]
  MoveL 3412 to (282.91, 241.46, -7.5) mm, rotated rx 180 ry 0 rz -180 deg; joints [-9.189, -42.604, 107.149, 169.843, 64.895, -175.653]
  MoveL 3413 to (283.39, 243.57, -7.5) mm, rotated rx 180 ry 0 rz 180 deg; joints [-9.265, -42.585, 107.095, 169.756, 64.865, -175.611]
  MoveL 3414 to (283.73, 245.7, -7.5) mm, rotated rx -180 ry 0 rz -180 deg; joints [-9.343, -42.57, 107.049, 169.668, 64.841, -175.568]
  MoveL 3415 to (283.93, 247.84, -7.5) mm, rotated rx 180 ry 0 rz -180 deg; joints [-9.421, -42.558, 107.012, 169.579, 64.823, -175.526]
  MoveL 3416 to (284, 250, -7.5) mm, rotated rx 180 ry 0 rz -180 deg; joints [-9.502, -42.548, 106.984, 169.489, 64.811, -175.485]
  MoveL 3417 to (272, 250, -7.5) mm, rotated rx -180 ry 0 rz 180 deg; joints [-9.577, -42.813, 107.779, 169.451, 65.338, -175.557]
  MoveL 3418 to (271.96, 251.4, -7.5) mm, rotated rx 180 ry 0 rz 180 deg; joints [-9.63, -42.809, 107.766, 169.393, 65.334, -175.531]
  MoveL 3419 to (271.82, 252.79, -7.5) mm, rotated rx 180 ry 0 rz -180 deg; joints [-9.683, -42.807, 107.759, 169.334, 65.333, -175.506]
  MoveL 3420 to (271.6, 254.16, -7.5) mm, rotated rx 180 ry 0 rz 180 deg; joints [-9.736, -42.807, 107.758, 169.276, 65.337, -175.481]
  MoveL 3421 to (271.29, 255.53, -7.5) mm, rotated rx -180 ry 0 rz 180 deg; joints [-9.789, -42.808, 107.763, 169.218, 65.344, -175.458]
  MoveL 3422 to (270.9, 256.86, -7.5) mm, rotated rx 180 ry 0 rz 180 deg; joints [-9.842, -42.812, 107.774, 169.16, 65.355, -175.435]
  MoveL 3423 to (270.42, 258.18, -7.5) mm, rotated rx -180 ry 0 rz 180 deg; joints [-9.894, -42.817, 107.79, 169.104, 65.37, -175.413]
  MoveL 3424 to (269.86, 259.46, -7.5) mm, rotated rx 180 ry 0 rz 180 deg; joints [-9.946, -42.825, 107.812, 169.048, 65.389, -175.393]
  MoveL 3425 to (269.22, 260.7, -7.5) mm, rotated rx -180 ry 0 rz -180 deg; joints [-9.997, -42.834, 107.84, 168.994, 65.411, -175.373]
  MoveL 3426 to (268.51, 261.89, -7.5) mm, rotated rx -180 ry 0 rz 180 deg; joints [-10.047, -42.845, 107.874, 168.942, 65.437, -175.355]
  MoveL 3427 to (267.72, 263.04, -7.5) mm, rotated rx 180 ry 0 rz -180 deg; joints [-10.095, -42.858, 107.912, 168.891, 65.467, -175.339]
  MoveL 3428 to (266.85, 264.14, -7.5) mm, rotated rx -180 ry 0 rz -180 deg; joints [-10.142, -42.872, 107.956, 168.842, 65.499, -175.324]
  MoveL 3429 to (265.92, 265.18, -7.5) mm, rotated rx 180 ry 0 rz -180 deg; joints [-10.188, -42.888, 108.005, 168.795, 65.535, -175.31]
  MoveL 3430 to (264.93, 266.16, -7.5) mm, rotated rx -180 ry 0 rz 180 deg; joints [-10.231, -42.906, 108.059, 168.75, 65.574, -175.298]
  MoveL 3431 to (263.87, 267.08, -7.5) mm, rotated rx -180 ry 0 rz 180 deg; joints [-10.273, -42.926, 108.118, 168.708, 65.616, -175.288]
  MoveL 3432 to (262.76, 267.92, -7.5) mm, rotated rx 180 ry 0 rz 180 deg; joints [-10.312, -42.946, 108.181, 168.669, 65.661, -175.279]
  MoveL 3433 to (261.6, 268.69, -7.5) mm, rotated rx 180 ry 0 rz -180 deg; joints [-10.35, -42.969, 108.248, 168.632, 65.708, -175.272]
  MoveL 3434 to (260.39, 269.39, -7.5) mm, rotated rx -180 ry 0 rz -180 deg; joints [-10.384, -42.992, 108.319, 168.599, 65.757, -175.267]
  MoveL 3435 to (259.14, 270.01, -7.5) mm, rotated rx -180 ry 0 rz -180 deg; joints [-10.416, -43.016, 108.394, 168.568, 65.809, -175.263]
  MoveL 3436 to (257.85, 270.55, -7.5) mm, rotated rx -180 ry 0 rz -180 deg; joints [-10.446, -43.042, 108.472, 168.541, 65.863, -175.261]
  MoveL 3437 to (256.53, 271.01, -7.5) mm, rotated rx 180 ry 0 rz 180 deg; joints [-10.472, -43.069, 108.553, 168.517, 65.918, -175.261]
  MoveL 3438 to (255.19, 271.38, -7.5) mm, rotated rx -180 ry 0 rz -180 deg; joints [-10.495, -43.096, 108.636, 168.496, 65.976, -175.263]
  MoveL 3439 to (253.82, 271.67, -7.5) mm, rotated rx -180 ry 0 rz -180 deg; joints [-10.516, -43.124, 108.722, 168.479, 66.034, -175.267]
  MoveL 3440 to (252.44, 271.86, -7.5) mm, rotated rx 180 ry 0 rz -180 deg; joints [-10.533, -43.153, 108.81, 168.466, 66.093, -175.272]
  MoveL 3441 to (251.05, 271.98, -7.5) mm, rotated rx -180 ry 0 rz -180 deg; joints [-10.547, -43.182, 108.9, 168.456, 66.154, -175.279]
  MoveL 3442 to (249.65, 272, -7.5) mm, rotated rx -180 ry 0 rz 180 deg; joints [-10.558, -43.212, 108.991, 168.449, 66.215, -175.288]
  MoveL 3443 to (248.26, 271.93, -7.5) mm, rotated rx 180 ry 0 rz -180 deg; joints [-10.565, -43.242, 109.083, 168.447, 66.276, -175.298]
  MoveL 3444 to (246.87, 271.78, -7.5) mm, rotated rx 180 ry 0 rz 180 deg; joints [-10.569, -43.272, 109.176, 168.448, 66.338, -175.31]
  MoveL 3445 to (245.49, 271.53, -7.5) mm, rotated rx 180 ry 0 rz -180 deg; joints [-10.57, -43.302, 109.268, 168.453, 66.399, -175.324]
  MoveL 3446 to (244.14, 271.2, -7.5) mm, rotated rx -180 ry 0 rz 180 deg; joints [-10.567, -43.332, 109.361, 168.462, 66.46, -175.339]
  MoveL 3447 to (242.8, 270.79, -7.5) mm, rotated rx -180 ry 0 rz -180 deg; joints [-10.56, -43.362, 109.453, 168.474, 66.521, -175.355]
  MoveL 3448 to (241.5, 270.29, -7.5) mm, rotated rx 180 ry 0 rz -180 deg; joints [-10.551, -43.391, 109.544, 168.49, 66.58, -175.373]
  MoveL 3449 to (240.23, 269.71, -7.5) mm, rotated rx 180 ry 0 rz 180 deg; joints [-10.538, -43.42, 109.634, 168.509, 66.639, -175.391]
  MoveL 3450 to (239, 269.05, -7.5) mm, rotated rx 180 ry 0 rz -180 deg; joints [-10.521, -43.448, 109.722, 168.532, 66.696, -175.412]
  MoveL 3451 to (237.81, 268.32, -7.5) mm, rotated rx -180 ry 0 rz -180 deg; joints [-10.501, -43.476, 109.808, 168.559, 66.752, -175.433]
  MoveL 3452 to (236.68, 267.51, -7.5) mm, rotated rx 180 ry 0 rz 180 deg; joints [-10.478, -43.503, 109.891, 168.588, 66.806, -175.455]
  MoveL 3453 to (235.59, 266.63, -7.5) mm, rotated rx -180 ry 0 rz -180 deg; joints [-10.452, -43.529, 109.972, 168.621, 66.858, -175.478]
  MoveL 3454 to (234.57, 265.68, -7.5) mm, rotated rx -180 ry 0 rz -180 deg; joints [-10.423, -43.554, 110.05, 168.657, 66.907, -175.501]
  MoveL 3455 to (233.6, 264.67, -7.5) mm, rotated rx 180 ry 0 rz -180 deg; joints [-10.391, -43.577, 110.125, 168.696, 66.955, -175.526]
  MoveL 3456 to (232.71, 263.6, -7.5) mm, rotated rx 180 ry 0 rz -180 deg; joints [-10.357, -43.6, 110.196, 168.738, 66.999, -175.551]
  MoveL 3457 to (231.88, 262.48, -7.5) mm, rotated rx 180 ry 0 rz -180 deg; joints [-10.319, -43.621, 110.263, 168.782, 67.041, -175.576]
  MoveL 3458 to (231.12, 261.3, -7.5) mm, rotated rx 180 ry 0 rz -180 deg; joints [-10.279, -43.641, 110.326, 168.829, 67.08, -175.602]
  MoveL 3459 to (230.45, 260.08, -7.5) mm, rotated rx 180 ry 0 rz -180 deg; joints [-10.237, -43.66, 110.384, 168.878, 67.116, -175.628]
  MoveL 3460 to (229.85, 258.82, -7.5) mm, rotated rx 180 ry 0 rz 180 deg; joints [-10.192, -43.677, 110.438, 168.929, 67.149, -175.655]
  MoveL 3461 to (229.33, 257.52, -7.5) mm, rotated rx -180 ry 0 rz -180 deg; joints [-10.146, -43.692, 110.487, 168.982, 67.178, -175.681]
  MoveL 3462 to (228.89, 256.2, -7.5) mm, rotated rx 180 ry 0 rz 180 deg; joints [-10.098, -43.706, 110.53, 169.036, 67.203, -175.707]
  MoveL 3463 to (228.54, 254.85, -7.5) mm, rotated rx -180 ry 0 rz 180 deg; joints [-10.048, -43.718, 110.568, 169.092, 67.225, -175.734]
  MoveL 3464 to (228.28, 253.48, -7.5) mm, rotated rx -180 ry 0 rz 180 deg; joints [-9.997, -43.729, 110.601, 169.149, 67.244, -175.76]
  MoveL 3465 to (228.1, 252.09, -7.5) mm, rotated rx 180 ry 0 rz 180 deg; joints [-9.945, -43.737, 110.629, 169.207, 67.258, -175.785]
  MoveL 3466 to (228.01, 250.7, -7.5) mm, rotated rx -180 ry 0 rz -180 deg; joints [-9.891, -43.744, 110.65, 169.266, 67.269, -175.811]
  MoveL 3467 to (228.01, 249.3, -7.5) mm, rotated rx 180 ry 0 rz -180 deg; joints [-9.837, -43.749, 110.666, 169.325, 67.275, -175.835]
  MoveL 3468 to (228.1, 247.91, -7.5) mm, rotated rx -180 ry 0 rz -180 deg; joints [-9.783, -43.752, 110.676, 169.385, 67.278, -175.859]
  MoveL 3469 to (228.28, 246.52, -7.5) mm, rotated rx -180 ry 0 rz -180 deg; joints [-9.728, -43.754, 110.68, 169.444, 67.277, -175.883]
  MoveL 3470 to (228.54, 245.15, -7.5) mm, rotated rx -180 ry 0 rz -180 deg; joints [-9.673, -43.753, 110.678, 169.503, 67.271, -175.905]
  MoveL 3471 to (228.89, 243.8, -7.5) mm, rotated rx -180 ry 0 rz 180 deg; joints [-9.619, -43.75, 110.67, 169.562, 67.262, -175.927]
  MoveL 3472 to (229.33, 242.48, -7.5) mm, rotated rx -180 ry 0 rz -180 deg; joints [-9.564, -43.746, 110.656, 169.62, 67.249, -175.948]
  MoveL 3473 to (229.85, 241.18, -7.5) mm, rotated rx -180 ry 0 rz 180 deg; joints [-9.511, -43.74, 110.637, 169.677, 67.232, -175.968]
  MoveL 3474 to (230.45, 239.92, -7.5) mm, rotated rx 180 ry 0 rz -180 deg; joints [-9.458, -43.732, 110.611, 169.733, 67.212, -175.987]
  MoveL 3475 to (231.12, 238.7, -7.5) mm, rotated rx 180 ry 0 rz 180 deg; joints [-9.407, -43.722, 110.58, 169.787, 67.187, -176.004]
  MoveL 3476 to (231.88, 237.52, -7.5) mm, rotated rx -180 ry 0 rz -180 deg; joints [-9.356, -43.711, 110.544, 169.839, 67.159, -176.02]
  MoveL 3477 to (232.71, 236.4, -7.5) mm, rotated rx 180 ry 0 rz 180 deg; joints [-9.308, -43.697, 110.502, 169.89, 67.128, -176.036]
  MoveL 3478 to (233.6, 235.33, -7.5) mm, rotated rx 180 ry 0 rz 180 deg; joints [-9.261, -43.683, 110.455, 169.939, 67.093, -176.049]
  MoveL 3479 to (234.57, 234.32, -7.5) mm, rotated rx -180 ry 0 rz -180 deg; joints [-9.215, -43.666, 110.403, 169.985, 67.055, -176.062]
  MoveL 3480 to (235.59, 233.37, -7.5) mm, rotated rx -180 ry 0 rz -180 deg; joints [-9.172, -43.648, 110.346, 170.029, 67.014, -176.072]
  MoveL 3481 to (236.68, 232.49, -7.5) mm, rotated rx -180 ry 0 rz -180 deg; joints [-9.132, -43.628, 110.285, 170.07, 66.97, -176.082]
  MoveL 3482 to (237.81, 231.68, -7.5) mm, rotated rx -180 ry 0 rz 180 deg; joints [-9.093, -43.608, 110.22, 170.108, 66.923, -176.09]
  MoveL 3483 to (239, 230.95, -7.5) mm, rotated rx -180 ry 0 rz 180 deg; joints [-9.058, -43.585, 110.15, 170.143, 66.874, -176.096]
  MoveL 3484 to (240.23, 230.29, -7.5) mm, rotated rx 180 ry 0 rz 180 deg; joints [-9.025, -43.562, 110.077, 170.175, 66.822, -176.101]
  MoveL 3485 to (241.5, 229.71, -7.5) mm, rotated rx -180 ry 0 rz -180 deg; joints [-8.995, -43.537, 110, 170.204, 66.769, -176.104]
  MoveL 3486 to (242.8, 229.21, -7.5) mm, rotated rx 180 ry 0 rz 180 deg; joints [-8.968, -43.512, 109.92, 170.23, 66.713, -176.106]
  MoveL 3487 to (244.14, 228.8, -7.5) mm, rotated rx 180 ry 0 rz 180 deg; joints [-8.943, -43.485, 109.837, 170.252, 66.656, -176.106]
  MoveL 3488 to (245.49, 228.47, -7.5) mm, rotated rx -180 ry 0 rz 180 deg; joints [-8.923, -43.458, 109.752, 170.27, 66.598, -176.104]
  MoveL 3489 to (246.87, 228.22, -7.5) mm, rotated rx 180 ry 0 rz 180 deg; joints [-8.905, -43.43, 109.664, 170.285, 66.538, -176.101]
  MoveL 3490 to (248.26, 228.07, -7.5) mm, rotated rx -180 ry 0 rz 180 deg; joints [-8.891, -43.401, 109.575, 170.296, 66.478, -176.096]
  MoveL 3491 to (249.65, 228, -7.5) mm, rotated rx -180 ry 0 rz 180 deg; joints [-8.88, -43.372, 109.484, 170.303, 66.416, -176.089]
  MoveL 3492 to (251.05, 228.02, -7.5) mm, rotated rx -180 ry 0 rz 180 deg; joints [-8.872, -43.342, 109.393, 170.307, 66.355, -176.081]
  MoveL 3493 to (252.44, 228.14, -7.5) mm, rotated rx -180 ry 0 rz -180 deg; joints [-8.868, -43.312, 109.3, 170.307, 66.293, -176.071]
  MoveL 3494 to (253.82, 228.33, -7.5) mm, rotated rx -180 ry 0 rz 180 deg; joints [-8.868, -43.282, 109.208, 170.303, 66.231, -176.06]
  MoveL 3495 to (255.19, 228.62, -7.5) mm, rotated rx 180 ry 0 rz 180 deg; joints [-8.87, -43.252, 109.115, 170.295, 66.17, -176.047]
  MoveL 3496 to (256.53, 228.99, -7.5) mm, rotated rx 180 ry 0 rz 180 deg; joints [-8.877, -43.222, 109.023, 170.284, 66.109, -176.033]
  MoveL 3497 to (257.85, 229.45, -7.5) mm, rotated rx 180 ry 0 rz 180 deg; joints [-8.886, -43.192, 108.931, 170.269, 66.049, -176.017]
  MoveL 3498 to (259.14, 229.99, -7.5) mm, rotated rx 180 ry 0 rz -180 deg; joints [-8.899, -43.163, 108.841, 170.25, 65.99, -176.001]
  MoveL 3499 to (260.39, 230.61, -7.5) mm, rotated rx -180 ry 0 rz -180 deg; joints [-8.915, -43.134, 108.753, 170.228, 65.932, -175.982]
  MoveL 3500 to (261.6, 231.31, -7.5) mm, rotated rx 180 ry 0 rz -180 deg; joints [-8.934, -43.106, 108.666, 170.202, 65.876, -175.963]
  MoveL 3501 to (262.76, 232.08, -7.5) mm, rotated rx -180 ry 0 rz -180 deg; joints [-8.957, -43.078, 108.581, 170.174, 65.821, -175.942]
  MoveL 3502 to (263.87, 232.92, -7.5) mm, rotated rx -180 ry 0 rz -180 deg; joints [-8.982, -43.051, 108.499, 170.142, 65.769, -175.92]
  MoveL 3503 to (264.93, 233.84, -7.5) mm, rotated rx -180 ry 0 rz 180 deg; joints [-9.011, -43.025, 108.42, 170.106, 65.718, -175.898]
  MoveL 3504 to (265.92, 234.82, -7.5) mm, rotated rx 180 ry 0 rz -180 deg; joints [-9.042, -43, 108.344, 170.068, 65.67, -175.874]
  MoveL 3505 to (266.85, 235.86, -7.5) mm, rotated rx -180 ry 0 rz -180 deg; joints [-9.076, -42.976, 108.272, 170.028, 65.625, -175.85]
  MoveL 3506 to (267.72, 236.96, -7.5) mm, rotated rx 180 ry 0 rz 180 deg; joints [-9.112, -42.954, 108.203, 169.984, 65.582, -175.824]
  MoveL 3507 to (268.51, 238.11, -7.5) mm, rotated rx -180 ry 0 rz -180 deg; joints [-9.15, -42.933, 108.139, 169.939, 65.543, -175.799]
  MoveL 3508 to (269.22, 239.3, -7.5) mm, rotated rx 180 ry 0 rz -180 deg; joints [-9.191, -42.913, 108.079, 169.891, 65.506, -175.772]
  MoveL 3509 to (269.86, 240.54, -7.5) mm, rotated rx -180 ry 0 rz -180 deg; joints [-9.234, -42.894, 108.023, 169.841, 65.473, -175.746]
  MoveL 3510 to (270.42, 241.82, -7.5) mm, rotated rx -180 ry 0 rz 180 deg; joints [-9.279, -42.878, 107.973, 169.789, 65.443, -175.719]
  MoveL 3511 to (270.9, 243.14, -7.5) mm, rotated rx -180 ry 0 rz -180 deg; joints [-9.326, -42.863, 107.927, 169.735, 65.416, -175.691]
  MoveL 3512 to (271.29, 244.47, -7.5) mm, rotated rx 180 ry 0 rz 180 deg; joints [-9.374, -42.849, 107.886, 169.68, 65.393, -175.664]
  MoveL 3513 to (271.6, 245.84, -7.5) mm, rotated rx 180 ry 0 rz 180 deg; joints [-9.423, -42.837, 107.851, 169.624, 65.373, -175.637]
  MoveL 3514 to (271.82, 247.22, -7.5) mm, rotated rx 180 ry 0 rz 180 deg; joints [-9.473, -42.828, 107.821, 169.567, 65.358, -175.61]
  MoveL 3515 to (271.96, 248.6, -7.5) mm, rotated rx -180 ry 0 rz 180 deg; joints [-9.525, -42.82, 107.797, 169.509, 65.346, -175.583]
  MoveL 3516 to (272, 250, -7.5) mm, rotated rx -180 ry 0 rz 180 deg; joints [-9.577, -42.813, 107.779, 169.451, 65.338, -175.557]
  MoveL 3517 to (260, 250, -7.5) mm, rotated rx -180 ry 0 rz -180 deg; joints [-9.654, -43.074, 108.57, 169.411, 65.865, -175.629]
  MoveL 3518 to (259.98, 250.63, -7.5) mm, rotated rx 180 ry 0 rz 180 deg; joints [-9.678, -43.072, 108.564, 169.385, 65.863, -175.617]
  MoveL 3519 to (259.92, 251.27, -7.5) mm, rotated rx 180 ry 0 rz 180 deg; joints [-9.702, -43.071, 108.561, 169.358, 65.863, -175.606]
  MoveL 3520 to (259.82, 251.89, -7.5) mm, rotated rx 180 ry 0 rz 180 deg; joints [-9.727, -43.071, 108.56, 169.331, 65.864, -175.595]
  MoveL 3521 to (259.68, 252.51, -7.5) mm, rotated rx -180 ry 0 rz -180 deg; joints [-9.751, -43.072, 108.563, 169.305, 65.867, -175.584]
  MoveL 3522 to (259.5, 253.12, -7.5) mm, rotated rx 180 ry 0 rz 180 deg; joints [-9.775, -43.074, 108.567, 169.278, 65.873, -175.574]
  MoveL 3523 to (259.28, 253.72, -7.5) mm, rotated rx 180 ry 0 rz -180 deg; joints [-9.799, -43.076, 108.575, 169.253, 65.879, -175.565]
  MoveL 3524 to (259.03, 254.3, -7.5) mm, rotated rx 180 ry 0 rz -180 deg; joints [-9.823, -43.079, 108.585, 169.227, 65.888, -175.555]
  MoveL 3525 to (258.74, 254.86, -7.5) mm, rotated rx 180 ry 0 rz -180 deg; joints [-9.846, -43.083, 108.598, 169.203, 65.898, -175.547]
  MoveL 3526 to (258.41, 255.41, -7.5) mm, rotated rx 180 ry 0 rz -180 deg; joints [-9.869, -43.088, 108.613, 169.179, 65.91, -175.539]
  MoveL 3527 to (258.05, 255.93, -7.5) mm, rotated rx 180 ry 0 rz -180 deg; joints [-9.891, -43.094, 108.631, 169.155, 65.923, -175.531]
  MoveL 3528 to (257.66, 256.43, -7.5) mm, rotated rx 180 ry 0 rz 180 deg; joints [-9.913, -43.101, 108.651, 169.133, 65.938, -175.525]
  MoveL 3529 to (257.24, 256.9, -7.5) mm, rotated rx 180 ry 0 rz -180 deg; joints [-9.933, -43.108, 108.673, 169.112, 65.955, -175.518]
  MoveL 3530 to (256.79, 257.35, -7.5) mm, rotated rx -180 ry 0 rz -180 deg; joints [-9.953, -43.116, 108.697, 169.091, 65.972, -175.513]
  MoveL 3531 to (256.31, 257.76, -7.5) mm, rotated rx 180 ry 0 rz 180 deg; joints [-9.972, -43.125, 108.724, 169.072, 65.991, -175.508]
  MoveL 3532 to (255.8, 258.15, -7.5) mm, rotated rx 180 ry 0 rz 180 deg; joints [-9.99, -43.134, 108.753, 169.054, 66.012, -175.504]
  MoveL 3533 to (255.27, 258.5, -7.5) mm, rotated rx -180 ry 0 rz -180 deg; joints [-10.007, -43.144, 108.783, 169.038, 66.033, -175.501]
  MoveL 3534 to (254.72, 258.81, -7.5) mm, rotated rx 180 ry 0 rz 180 deg; joints [-10.023, -43.155, 108.816, 169.022, 66.056, -175.499]
  MoveL 3535 to (254.15, 259.1, -7.5) mm, rotated rx -180 ry 0 rz -180 deg; joints [-10.037, -43.166, 108.85, 169.009, 66.08, -175.497]
  MoveL 3536 to (253.57, 259.34, -7.5) mm, rotated rx -180 ry 0 rz -180 deg; joints [-10.05, -43.177, 108.885, 168.996, 66.104, -175.496]
  MoveL 3537 to (252.97, 259.55, -7.5) mm, rotated rx 180 ry 0 rz -180 deg; joints [-10.062, -43.189, 108.922, 168.985, 66.129, -175.496]
  MoveL 3538 to (252.36, 259.72, -7.5) mm, rotated rx -180 ry 0 rz 180 deg; joints [-10.073, -43.202, 108.96, 168.976, 66.156, -175.497]
  MoveL 3539 to (251.74, 259.85, -7.5) mm, rotated rx -180 ry 0 rz -180 deg; joints [-10.082, -43.215, 108.999, 168.968, 66.182, -175.498]
  MoveL 3540 to (251.11, 259.94, -7.5) mm, rotated rx -180 ry 0 rz -180 deg; joints [-10.09, -43.228, 109.04, 168.962, 66.209, -175.501]
  MoveL 3541 to (250.48, 259.99, -7.5) mm, rotated rx 180 ry 0 rz 180 deg; joints [-10.096, -43.241, 109.08, 168.958, 66.237, -175.504]
  MoveL 3542 to (249.84, 260, -7.5) mm, rotated rx -180 ry 0 rz 180 deg; joints [-10.101, -43.254, 109.122, 168.955, 66.265, -175.508]
  MoveL 3543 to (249.21, 259.97, -7.5) mm, rotated rx -180 ry 0 rz -180 deg; joints [-10.104, -43.268, 109.164, 168.954, 66.293, -175.512]
  MoveL 3544 to (248.58, 259.9, -7.5) mm, rotated rx 180 ry 0 rz -180 deg; joints [-10.105, -43.282, 109.206, 168.955, 66.321, -175.517]
  MoveL 3545 to (247.95, 259.79, -7.5) mm, rotated rx 180 ry 0 rz 180 deg; joints [-10.105, -43.295, 109.248, 168.957, 66.349, -175.523]
  MoveL 3546 to (247.34, 259.64, -7.5) mm, rotated rx -180 ry 0 rz 180 deg; joints [-10.104, -43.309, 109.29, 168.961, 66.376, -175.53]
  MoveL 3547 to (246.73, 259.45, -7.5) mm, rotated rx 180 ry 0 rz -180 deg; joints [-10.101, -43.322, 109.332, 168.967, 66.404, -175.537]
  MoveL 3548 to (246.14, 259.22, -7.5) mm, rotated rx 180 ry 0 rz -180 deg; joints [-10.096, -43.336, 109.373, 168.974, 66.431, -175.545]
  MoveL 3549 to (245.56, 258.96, -7.5) mm, rotated rx 180 ry 0 rz -180 deg; joints [-10.09, -43.349, 109.414, 168.983, 66.457, -175.553]
  MoveL 3550 to (245, 258.66, -7.5) mm, rotated rx 180 ry 0 rz -180 deg; joints [-10.082, -43.362, 109.454, 168.993, 66.483, -175.562]
  MoveL 3551 to (244.46, 258.33, -7.5) mm, rotated rx -180 ry 0 rz -180 deg; joints [-10.073, -43.374, 109.493, 169.006, 66.509, -175.572]
  MoveL 3552 to (243.94, 257.96, -7.5) mm, rotated rx 180 ry 0 rz 180 deg; joints [-10.063, -43.387, 109.531, 169.019, 66.533, -175.582]
  MoveL 3553 to (243.45, 257.56, -7.5) mm, rotated rx -180 ry 0 rz 180 deg; joints [-10.051, -43.399, 109.567, 169.034, 66.557, -175.592]
  MoveL 3554 to (242.99, 257.13, -7.5) mm, rotated rx -180 ry 0 rz -180 deg; joints [-10.037, -43.41, 109.603, 169.051, 66.579, -175.603]
  MoveL 3555 to (242.55, 256.67, -7.5) mm, rotated rx -180 ry 0 rz -180 deg; joints [-10.023, -43.421, 109.637, 169.068, 66.601, -175.614]
  MoveL 3556 to (242.14, 256.18, -7.5) mm, rotated rx 180 ry 0 rz -180 deg; joints [-10.007, -43.431, 109.669, 169.087, 66.621, -175.625]
  MoveL 3557 to (241.76, 255.67, -7.5) mm, rotated rx -180 ry 0 rz -180 deg; joints [-9.99, -43.441, 109.699, 169.108, 66.64, -175.637]
  MoveL 3558 to (241.42, 255.14, -7.5) mm, rotated rx 180 ry 0 rz 180 deg; joints [-9.972, -43.45, 109.728, 169.129, 66.657, -175.648]
  MoveL 3559 to (241.11, 254.58, -7.5) mm, rotated rx -180 ry 0 rz 180 deg; joints [-9.953, -43.459, 109.754, 169.151, 66.674, -175.66]
  MoveL 3560 to (240.84, 254.01, -7.5) mm, rotated rx -180 ry 0 rz 180 deg; joints [-9.933, -43.466, 109.779, 169.174, 66.688, -175.672]
  MoveL 3561 to (240.6, 253.42, -7.5) mm, rotated rx -180 ry 0 rz -180 deg; joints [-9.912, -43.474, 109.801, 169.198, 66.701, -175.685]
  MoveL 3562 to (240.41, 252.82, -7.5) mm, rotated rx -180 ry 0 rz 180 deg; joints [-9.89, -43.48, 109.82, 169.223, 66.713, -175.697]
  MoveL 3563 to (240.25, 252.2, -7.5) mm, rotated rx 180 ry 0 rz -180 deg; joints [-9.867, -43.485, 109.838, 169.248, 66.723, -175.709]
  MoveL 3564 to (240.13, 251.58, -7.5) mm, rotated rx -180 ry 0 rz 180 deg; joints [-9.844, -43.49, 109.853, 169.274, 66.731, -175.721]
  MoveL 3565 to (240.05, 250.95, -7.5) mm, rotated rx -180 ry 0 rz 180 deg; joints [-9.821, -43.494, 109.865, 169.301, 66.738, -175.732]
  MoveL 3566 to (240.01, 250.32, -7.5) mm, rotated rx 180 ry 0 rz 180 deg; joints [-9.797, -43.497, 109.875, 169.327, 66.742, -175.744]
  MoveL 3567 to (240.01, 249.68, -7.5) mm, rotated rx 180 ry 0 rz 180 deg; joints [-9.772, -43.5, 109.882, 169.354, 66.745, -175.756]
  MoveL 3568 to (240.05, 249.05, -7.5) mm, rotated rx 180 ry 0 rz 180 deg; joints [-9.748, -43.501, 109.886, 169.381, 66.746, -175.767]
  MoveL 3569 to (240.13, 248.42, -7.5) mm, rotated rx -180 ry 0 rz 180 deg; joints [-9.723, -43.502, 109.888, 169.408, 66.746, -175.777]
  MoveL 3570 to (240.25, 247.8, -7.5) mm, rotated rx 180 ry 0 rz 180 deg; joints [-9.698, -43.501, 109.887, 169.435, 66.743, -175.788]
  MoveL 3571 to (240.41, 247.18, -7.5) mm, rotated rx -180 ry 0 rz 180 deg; joints [-9.674, -43.5, 109.884, 169.461, 66.739, -175.798]
  MoveL 3572 to (240.6, 246.58, -7.5) mm, rotated rx -180 ry 0 rz -180 deg; joints [-9.649, -43.498, 109.878, 169.487, 66.733, -175.808]
  MoveL 3573 to (240.84, 245.99, -7.5) mm, rotated rx -180 ry 0 rz -180 deg; joints [-9.625, -43.495, 109.869, 169.513, 66.726, -175.817]
  MoveL 3574 to (241.11, 245.42, -7.5) mm, rotated rx 180 ry 0 rz 180 deg; joints [-9.601, -43.492, 109.857, 169.538, 66.716, -175.825]
  MoveL 3575 to (241.42, 244.86, -7.5) mm, rotated rx 180 ry 0 rz 180 deg; joints [-9.578, -43.487, 109.843, 169.563, 66.705, -175.834]
  MoveL 3576 to (241.76, 244.33, -7.5) mm, rotated rx 180 ry 0 rz -180 deg; joints [-9.555, -43.482, 109.827, 169.587, 66.693, -175.841]
  MoveL 3577 to (242.14, 243.82, -7.5) mm, rotated rx 180 ry 0 rz -180 deg; joints [-9.533, -43.476, 109.808, 169.61, 66.678, -175.848]
  MoveL 3578 to (242.55, 243.33, -7.5) mm, rotated rx 180 ry 0 rz 180 deg; joints [-9.512, -43.469, 109.786, 169.632, 66.663, -175.854]
  MoveL 3579 to (242.99, 242.87, -7.5) mm, rotated rx 180 ry 0 rz 180 deg; joints [-9.491, -43.461, 109.763, 169.653, 66.645, -175.86]
  MoveL 3580 to (243.45, 242.44, -7.5) mm, rotated rx 180 ry 0 rz -180 deg; joints [-9.472, -43.453, 109.737, 169.672, 66.627, -175.865]
  MoveL 3581 to (243.94, 242.04, -7.5) mm, rotated rx 180 ry 0 rz -180 deg; joints [-9.453, -43.444, 109.709, 169.691, 66.607, -175.869]
  MoveL 3582 to (244.46, 241.67, -7.5) mm, rotated rx -180 ry 0 rz 180 deg; joints [-9.436, -43.435, 109.68, 169.708, 66.586, -175.873]
  MoveL 3583 to (245, 241.34, -7.5) mm, rotated rx -180 ry 0 rz -180 deg; joints [-9.42, -43.424, 109.648, 169.724, 66.563, -175.876]
  MoveL 3584 to (245.56, 241.04, -7.5) mm, rotated rx -180 ry 0 rz -180 deg; joints [-9.405, -43.414, 109.615, 169.739, 66.54, -175.878]
  MoveL 3585 to (246.14, 240.78, -7.5) mm, rotated rx -180 ry 0 rz 180 deg; joints [-9.391, -43.403, 109.58, 169.752, 66.516, -175.879]
  MoveL 3586 to (246.73, 240.55, -7.5) mm, rotated rx 180 ry 0 rz 180 deg; joints [-9.379, -43.391, 109.544, 169.764, 66.491, -175.88]
  MoveL 3587 to (247.34, 240.36, -7.5) mm, rotated rx -180 ry 0 rz -180 deg; joints [-9.368, -43.379, 109.506, 169.774, 66.465, -175.88]
  MoveL 3588 to (247.95, 240.21, -7.5) mm, rotated rx -180 ry 0 rz -180 deg; joints [-9.358, -43.366, 109.467, 169.782, 66.438, -175.879]
  MoveL 3589 to (248.58, 240.1, -7.5) mm, rotated rx -180 ry 0 rz 180 deg; joints [-9.35, -43.353, 109.428, 169.789, 66.411, -175.877]
  MoveL 3590 to (249.21, 240.03, -7.5) mm, rotated rx -180 ry 0 rz -180 deg; joints [-9.343, -43.34, 109.387, 169.794, 66.384, -175.875]
  MoveL 3591 to (249.84, 240, -7.5) mm, rotated rx 180 ry 0 rz 180 deg; joints [-9.338, -43.327, 109.346, 169.798, 66.356, -175.872]
  MoveL 3592 to (250.48, 240.01, -7.5) mm, rotated rx 180 ry 0 rz -180 deg; joints [-9.334, -43.314, 109.304, 169.799, 66.328, -175.868]
  MoveL 3593 to (251.11, 240.06, -7.5) mm, rotated rx -180 ry 0 rz -180 deg; joints [-9.332, -43.3, 109.262, 169.799, 66.3, -175.863]
  MoveL 3594 to (251.74, 240.15, -7.5) mm, rotated rx -180 ry 0 rz -180 deg; joints [-9.332, -43.286, 109.22, 169.798, 66.272, -175.858]
  MoveL 3595 to (252.36, 240.28, -7.5) mm, rotated rx 180 ry 0 rz -180 deg; joints [-9.333, -43.273, 109.178, 169.794, 66.244, -175.852]
  MoveL 3596 to (252.97, 240.45, -7.5) mm, rotated rx 180 ry 0 rz 180 deg; joints [-9.335, -43.259, 109.136, 169.789, 66.216, -175.845]
  MoveL 3597 to (253.57, 240.66, -7.5) mm, rotated rx 180 ry 0 rz 180 deg; joints [-9.34, -43.245, 109.095, 169.783, 66.189, -175.838]
  MoveL 3598 to (254.15, 240.9, -7.5) mm, rotated rx 180 ry 0 rz -180 deg; joints [-9.345, -43.232, 109.054, 169.774, 66.162, -175.83]
  MoveL 3599 to (254.72, 241.19, -7.5) mm, rotated rx 180 ry 0 rz 180 deg; joints [-9.352, -43.219, 109.013, 169.764, 66.136, -175.822]
  MoveL 3600 to (255.27, 241.5, -7.5) mm, rotated rx 180 ry 0 rz -180 deg; joints [-9.361, -43.206, 108.974, 169.753, 66.11, -175.813]
  MoveL 3601 to (255.8, 241.85, -7.5) mm, rotated rx -180 ry 0 rz -180 deg; joints [-9.371, -43.194, 108.935, 169.74, 66.086, -175.803]
  MoveL 3602 to (256.31, 242.24, -7.5) mm, rotated rx -180 ry 0 rz 180 deg; joints [-9.383, -43.182, 108.898, 169.725, 66.062, -175.793]
  MoveL 3603 to (256.79, 242.65, -7.5) mm, rotated rx 180 ry 0 rz -180 deg; joints [-9.395, -43.17, 108.862, 169.709, 66.039, -175.783]
  MoveL 3604 to (257.24, 243.1, -7.5) mm, rotated rx -180 ry 0 rz -180 deg; joints [-9.409, -43.159, 108.827, 169.692, 66.017, -175.772]
  MoveL 3605 to (257.66, 243.57, -7.5) mm, rotated rx -180 ry 0 rz -180 deg; joints [-9.425, -43.148, 108.794, 169.674, 65.996, -175.761]
  MoveL 3606 to (258.05, 244.07, -7.5) mm, rotated rx -180 ry 0 rz 180 deg; joints [-9.441, -43.138, 108.763, 169.654, 65.977, -175.749]
  MoveL 3607 to (258.41, 244.59, -7.5) mm, rotated rx -180 ry 0 rz -180 deg; joints [-9.459, -43.128, 108.734, 169.633, 65.959, -175.738]
  MoveL 3608 to (258.74, 245.14, -7.5) mm, rotated rx -180 ry 0 rz 180 deg; joints [-9.477, -43.119, 108.706, 169.611, 65.942, -175.726]
  MoveL 3609 to (259.03, 245.7, -7.5) mm, rotated rx -180 ry 0 rz 180 deg; joints [-9.497, -43.111, 108.681, 169.589, 65.927, -175.714]
  MoveL 3610 to (259.28, 246.28, -7.5) mm, rotated rx -180 ry 0 rz -180 deg; joints [-9.517, -43.103, 108.658, 169.565, 65.913, -175.702]
  MoveL 3611 to (259.5, 246.88, -7.5) mm, rotated rx 180 ry 0 rz -180 deg; joints [-9.539, -43.096, 108.637, 169.541, 65.901, -175.689]
  MoveL 3612 to (259.68, 247.49, -7.5) mm, rotated rx 180 ry 0 rz 180 deg; joints [-9.561, -43.09, 108.619, 169.516, 65.89, -175.677]
  MoveL 3613 to (259.82, 248.11, -7.5) mm, rotated rx 180 ry 0 rz 180 deg; joints [-9.583, -43.085, 108.603, 169.49, 65.881, -175.665]
  MoveL 3614 to (259.92, 248.73, -7.5) mm, rotated rx 180 ry 0 rz -180 deg; joints [-9.606, -43.081, 108.589, 169.464, 65.874, -175.653]
  MoveL 3615 to (259.98, 249.37, -7.5) mm, rotated rx -180 ry 0 rz -180 deg; joints [-9.63, -43.077, 108.578, 169.438, 65.868, -175.641]
  MoveL 3616 to (260, 250, -7.5) mm, rotated rx -180 ry 0 rz -180 deg; joints [-9.654, -43.074, 108.57, 169.411, 65.865, -175.629]
  Establecer velocidad (1000.0 mm/s)
  MoveL 3617 to (260, 250, 10) mm, rotated rx 180 ry 0 rz -180 deg; joints [-9.654, -44.022, 108.777, 169.349, 65.137, -175.479]
  MoveL 3618 to (392, 250, 10) mm, rotated rx -180 ry 0 rz -180 deg; joints [-8.871, -40.818, 99.818, 169.68, 59.411, -174.706]
  MoveL 3619 to (392, 250, 10) mm, rotated rx -180 ry 0 rz -180 deg; joints [-8.871, -40.818, 99.818, 169.68, 59.411, -174.706]
  MoveL 3620 to (392, 250, 10) mm, rotated rx -180 ry 0 rz -180 deg; joints [-8.871, -40.818, 99.818, 169.68, 59.411, -174.706]
  Establecer velocidad (1.7 mm/s)
  MoveL 3621 to (392, 250, -10) mm, rotated rx 180 ry 0 rz -180 deg; joints [-8.871, -39.832, 99.591, 169.759, 60.157, -174.863]
  Establecer velocidad (16.7 mm/s)
  MoveL 3622 to (392, 250, -10) mm, rotated rx 180 ry 0 rz -180 deg; joints [-8.871, -39.832, 99.591, 169.759, 60.157, -174.863]
  MoveL 3623 to (391.71, 259.01, -10) mm, rotated rx 180 ry 0 rz 180 deg; joints [-9.187, -39.803, 99.51, 169.391, 60.136, -174.671]
  MoveL 3624 to (390.86, 267.98, -10) mm, rotated rx 180 ry 0 rz -180 deg; joints [-9.505, -39.787, 99.467, 169.023, 60.139, -174.484]
  MoveL 3625 to (389.43, 276.87, -10) mm, rotated rx -180 ry 0 rz -180 deg; joints [-9.823, -39.785, 99.461, 168.658, 60.166, -174.301]
  MoveL 3626 to (387.45, 285.66, -10) mm, rotated rx -180 ry 0 rz -180 deg; joints [-10.141, -39.796, 99.491, 168.296, 60.217, -174.125]
  MoveL 3627 to (384.91, 294.31, -10) mm, rotated rx 180 ry 0 rz -180 deg; joints [-10.457, -39.821, 99.559, 167.938, 60.292, -173.955]
  MoveL 3628 to (381.83, 302.78, -10) mm, rotated rx 180 ry 0 rz 180 deg; joints [-10.771, -39.859, 99.663, 167.587, 60.39, -173.793]
  MoveL 3629 to (378.22, 311.03, -10) mm, rotated rx 180 ry 0 rz -180 deg; joints [-11.082, -39.91, 99.803, 167.242, 60.511, -173.64]
  MoveL 3630 to (374.09, 319.04, -10) mm, rotated rx -180 ry 0 rz 180 deg; joints [-11.389, -39.974, 99.979, 166.906, 60.654, -173.497]
  MoveL 3631 to (369.46, 326.77, -10) mm, rotated rx 180 ry 0 rz 180 deg; joints [-11.691, -40.051, 100.19, 166.58, 60.819, -173.364]
  MoveL 3632 to (364.35, 334.19, -10) mm, rotated rx 180 ry 0 rz 180 deg; joints [-11.987, -40.14, 100.436, 166.264, 61.006, -173.243]
  MoveL 3633 to (358.78, 341.28, -10) mm, rotated rx 180 ry 0 rz -180 deg; joints [-12.275, -40.241, 100.714, 165.96, 61.212, -173.134]
  MoveL 3634 to (352.77, 347.99, -10) mm, rotated rx -180 ry 0 rz 180 deg; joints [-12.556, -40.353, 101.025, 165.67, 61.439, -173.037]
  MoveL 3635 to (346.35, 354.31, -10) mm, rotated rx 180 ry 0 rz 180 deg; joints [-12.828, -40.476, 101.366, 165.393, 61.684, -172.953]
  MoveL 3636 to (339.54, 360.21, -10) mm, rotated rx -180 ry 0 rz -180 deg; joints [-13.089, -40.609, 101.738, 165.13, 61.946, -172.882]
  MoveL 3637 to (332.37, 365.67, -10) mm, rotated rx 180 ry 0 rz -180 deg; joints [-13.34, -40.751, 102.137, 164.884, 62.226, -172.826]
  MoveL 3638 to (324.87, 370.66, -10) mm, rotated rx -180 ry 0 rz 180 deg; joints [-13.579, -40.903, 102.564, 164.654, 62.521, -172.783]
  MoveL 3639 to (317.06, 375.17, -10) mm, rotated rx -180 ry 0 rz -180 deg; joints [-13.806, -41.062, 103.015, 164.441, 62.831, -172.755]
  MoveL 3640 to (308.99, 379.17, -10) mm, rotated rx -180 ry 0 rz 180 deg; joints [-14.018, -41.229, 103.49, 164.247, 63.155, -172.74]
  MoveL 3641 to (300.68, 382.65, -10) mm, rotated rx -180 ry 0 rz -180 deg; joints [-14.217, -41.402, 103.986, 164.071, 63.49, -172.74]
  MoveL 3642 to (292.16, 385.6, -10) mm, rotated rx -180 ry 0 rz -180 deg; joints [-14.399, -41.581, 104.502, 163.915, 63.837, -172.754]
  MoveL 3643 to (283.48, 388, -10) mm, rotated rx -180 ry 0 rz -180 deg; joints [-14.566, -41.765, 105.036, 163.778, 64.194, -172.782]
  MoveL 3644 to (274.66, 389.84, -10) mm, rotated rx 180 ry 0 rz 180 deg; joints [-14.715, -41.953, 105.585, 163.662, 64.56, -172.823]
  MoveL 3645 to (265.74, 391.13, -10) mm, rotated rx 180 ry 0 rz 180 deg; joints [-14.847, -42.144, 106.148, 163.568, 64.933, -172.877]
  MoveL 3646 to (256.76, 391.84, -10) mm, rotated rx -180 ry 0 rz 180 deg; joints [-14.96, -42.337, 106.722, 163.494, 65.312, -172.944]
  MoveL 3647 to (247.75, 391.98, -10) mm, rotated rx 180 ry 0 rz -180 deg; joints [-15.054, -42.532, 107.305, 163.442, 65.696, -173.024]
  MoveL 3648 to (238.75, 391.55, -10) mm, rotated rx 180 ry 0 rz 180 deg; joints [-15.127, -42.728, 107.896, 163.413, 66.083, -173.114]
  MoveL 3649 to (229.79, 390.55, -10) mm, rotated rx 180 ry 0 rz 180 deg; joints [-15.18, -42.923, 108.491, 163.406, 66.473, -173.216]
  MoveL 3650 to (220.92, 388.99, -10) mm, rotated rx -180 ry 0 rz 180 deg; joints [-15.211, -43.117, 109.088, 163.422, 66.863, -173.328]
  MoveL 3651 to (212.16, 386.87, -10) mm, rotated rx -180 ry 0 rz -180 deg; joints [-15.221, -43.309, 109.685, 163.46, 67.252, -173.449]
  MoveL 3652 to (203.56, 384.19, -10) mm, rotated rx 180 ry 0 rz 180 deg; joints [-15.208, -43.498, 110.28, 163.522, 67.64, -173.579]
  MoveL 3653 to (195.14, 380.97, -10) mm, rotated rx -180 ry 0 rz -180 deg; joints [-15.173, -43.684, 110.87, 163.606, 68.023, -173.717]
  MoveL 3654 to (186.94, 377.23, -10) mm, rotated rx -180 ry 0 rz 180 deg; joints [-15.115, -43.866, 111.453, 163.713, 68.402, -173.862]
  MoveL 3655 to (179, 372.98, -10) mm, rotated rx 180 ry 0 rz -180 deg; joints [-15.034, -44.042, 112.026, 163.843, 68.775, -174.013]
  MoveL 3656 to (171.34, 368.22, -10) mm, rotated rx -180 ry 0 rz -180 deg; joints [-14.929, -44.213, 112.588, 163.996, 69.139, -174.168]
  MoveL 3657 to (164, 363, -10) mm, rotated rx 180 ry 0 rz -180 deg; joints [-14.802, -44.378, 113.135, 164.171, 69.495, -174.328]
  MoveL 3658 to (157.01, 357.32, -10) mm, rotated rx 180 ry 0 rz 180 deg; joints [-14.652, -44.536, 113.666, 164.368, 69.839, -174.492]
  MoveL 3659 to (150.39, 351.2, -10) mm, rotated rx 180 ry 0 rz 180 deg; joints [-14.479, -44.687, 114.179, 164.587, 70.171, -174.657]
  MoveL 3660 to (144.17, 344.68, -10) mm, rotated rx 180 ry 0 rz 180 deg; joints [-14.283, -44.829, 114.67, 164.826, 70.49, -174.824]
  MoveL 3661 to (138.38, 337.78, -10) mm, rotated rx -180 ry 0 rz -180 deg; joints [-14.067, -44.964, 115.138, 165.086, 70.793, -174.992]
  MoveL 3662 to (133.04, 330.52, -10) mm, rotated rx -180 ry 0 rz 180 deg; joints [-13.829, -45.09, 115.582, 165.364, 71.079, -175.16]
  MoveL 3663 to (128.17, 322.94, -10) mm, rotated rx 180 ry 0 rz 180 deg; joints [-13.571, -45.207, 115.998, 165.661, 71.348, -175.326]
  MoveL 3664 to (123.79, 315.07, -10) mm, rotated rx 180 ry 0 rz 180 deg; joints [-13.294, -45.314, 116.386, 165.976, 71.597, -175.491]
  MoveL 3665 to (119.91, 306.93, -10) mm, rotated rx -180 ry 0 rz 180 deg; joints [-12.999, -45.412, 116.743, 166.306, 71.826, -175.654]
  MoveL 3666 to (116.56, 298.57, -10) mm, rotated rx 180 ry 0 rz -180 deg; joints [-12.687, -45.501, 117.067, 166.651, 72.032, -175.813]
  MoveL 3667 to (113.75, 290.01, -10) mm, rotated rx -180 ry 0 rz -180 deg; joints [-12.36, -45.579, 117.358, 167.009, 72.216, -175.969]
  MoveL 3668 to (111.49, 281.28, -10) mm, rotated rx -180 ry 0 rz -180 deg; joints [-12.019, -45.648, 117.615, 167.38, 72.375, -176.122]
  MoveL 3669 to (109.78, 272.44, -10) mm, rotated rx -180 ry 0 rz -180 deg; joints [-11.666, -45.706, 117.834, 167.76, 72.509, -176.27]
  MoveL 3670 to (108.64, 263.5, -10) mm, rotated rx -180 ry 0 rz -180 deg; joints [-11.303, -45.754, 118.017, 168.149, 72.618, -176.413]
  MoveL 3671 to (108.07, 254.51, -10) mm, rotated rx -180 ry 0 rz -180 deg; joints [-10.931, -45.792, 118.161, 168.544, 72.699, -176.551]
